   LaserEnd_Ext()
   LIN {X -2.280, Y -28.706, Z 16.150}
   LaserStart_Ext()
   LIN {X -2.280, Y -30.758, Z 16.150}
   LaserEnd_Ext()
   LIN {X -1.280, Y -30.373, Z 16.150}
   LaserStart_Ext()
   LIN {X -1.280, Y -28.244, Z 16.150}
   LaserEnd_Ext()
   LIN {X -1.280, Y -17.881, Z 16.150}
   LaserStart_Ext()
   LIN {X -1.280, Y 7.950, Z 16.150}
   LaserEnd_Ext()
   LIN {X -1.280, Y 30.841, Z 16.150}
   LaserStart_Ext()
   LIN {X -1.280, Y 40.883, Z 16.150}
   LaserEnd_Ext()
   LIN {X -0.280, Y 41.227, Z 16.150}
   LaserStart_Ext()
   LIN {X -0.280, Y -18.756, Z 16.150}
   LaserEnd_Ext()
   LIN {X -0.280, Y -27.386, Z 16.150}
   LaserStart_Ext()
   LIN {X -0.280, Y -29.936, Z 16.150}
   LaserEnd_Ext()
   LIN {X 0.720, Y -29.192, Z 16.150}
   LaserStart_Ext()
   LIN {X 0.720, Y -26.394, Z 16.150}
   LaserEnd_Ext()
   LIN {X 0.720, Y -19.688, Z 16.150}
   LaserStart_Ext()
   LIN {X 0.720, Y 41.215, Z 16.150}
   LaserEnd_Ext()
   LIN {X 1.720, Y 40.867, Z 16.150}
   LaserStart_Ext()
   LIN {X 1.720, Y -23.022, Z 16.150}
   LaserEnd_Ext()
   LIN {X 1.720, Y -23.653, Z 16.150}
   LaserStart_Ext()
   LIN {X 1.720, Y -28.282, Z 16.150}
   LaserEnd_Ext()
   LIN {X 2.720, Y -26.691, Z 16.150}
   LaserStart_Ext()
   LIN {X 2.720, Y 39.894, Z 16.150}
   LaserEnd_Ext()
   LIN {X 3.720, Y 37.137, Z 16.150}
   LaserStart_Ext()
   LIN {X 3.720, Y -24.352, Z 16.150}
   LaserEnd_Ext()
   LIN {X 4.720, Y -20.713, Z 16.150}
   LaserStart_Ext()
   LIN {X 4.720, Y 33.485, Z 16.150}
   LaserEnd_Ext()
   LIN {X 5.720, Y 29.196, Z 16.150}
   LaserStart_Ext()
   LIN {X 5.720, Y -16.461, Z 16.150}
   LaserEnd_Ext()
   LIN {X 6.720, Y -11.133, Z 16.150}
   LaserStart_Ext()
   LIN {X 6.720, Y 23.723, Z 16.150}
   LaserEnd_Ext()
   LIN {X 7.720, Y 15.659, Z 16.150}
   LaserStart_Ext()
   LIN {X 7.720, Y -3.019, Z 16.150}
   LaserEnd_Ext()
   LIN {X -5.450, Y -18.220, Z 17.000}
   LaserStart_Ext()
   LIN {X -4.243, Y -18.029, Z 17.000} C_DIS
   LIN {X -3.691, Y -18.103, Z 17.000} C_DIS
   LIN {X -1.993, Y -18.493, Z 17.000} C_DIS
   LIN {X -0.415, Y -19.723, Z 17.000} C_DIS
   LIN {X -0.294, Y -19.833, Z 17.000} C_DIS
   LIN {X 0.476, Y -21.132, Z 17.000} C_DIS
   LIN {X 0.538, Y -21.297, Z 17.000} C_DIS
   LIN {X 0.796, Y -22.497, Z 17.000} C_DIS
   LIN {X 0.823, Y -23.103, Z 17.000} C_DIS
   LIN {X 0.725, Y -23.910, Z 17.000} C_DIS
   LIN {X 0.164, Y -25.394, Z 17.000} C_DIS
   LIN {X -0.518, Y -26.215, Z 17.000} C_DIS
   LIN {X -2.057, Y -27.540, Z 17.000} C_DIS
   LIN {X -3.374, Y -27.928, Z 17.000} C_DIS
   LIN {X -3.846, Y -28.000, Z 17.000} C_DIS
   LIN {X -4.662, Y -27.994, Z 17.000} C_DIS
   LIN {X -5.636, Y -27.809, Z 17.000} C_DIS
   LIN {X -6.024, Y -27.663, Z 17.000} C_DIS
   LIN {X -6.355, Y -27.534, Z 17.000} C_DIS
   LIN {X -6.753, Y -27.306, Z 17.000} C_DIS
   LIN {X -6.978, Y -27.176, Z 17.000} C_DIS
   LIN {X -7.114, Y -27.065, Z 17.000} C_DIS
   LIN {X -7.700, Y -26.583, Z 17.000} C_DIS
   LIN {X -7.930, Y -26.330, Z 17.000} C_DIS
   LIN {X -8.121, Y -26.097, Z 17.000} C_DIS
   LIN {X -8.706, Y -25.137, Z 17.000} C_DIS
   LIN {X -8.894, Y -24.608, Z 17.000} C_DIS
   LIN {X -9.152, Y -23.495, Z 17.000} C_DIS
   LIN {X -9.139, Y -22.986, Z 17.000} C_DIS
   LIN {X -8.912, Y -21.521, Z 17.000} C_DIS
   LIN {X -8.559, Y -20.716, Z 17.000} C_DIS
   LIN {X -7.683, Y -19.537, Z 17.000} C_DIS
   LIN {X -6.841, Y -18.853, Z 17.000} C_DIS
   LIN {X -5.450, Y -18.220, Z 17.000}
   LaserEnd_Ext()
   LIN {X 6.431, Y 30.497, Z 17.000}
   LaserStart_Ext()
   LIN {X 6.704, Y 29.214, Z 17.000} C_DIS
   LIN {X 6.976, Y 27.929, Z 17.000} C_DIS
   LIN {X 7.359, Y 25.908, Z 17.000} C_DIS
   LIN {X 8.015, Y 21.716, Z 17.000} C_DIS
   LIN {X 8.202, Y 20.509, Z 17.000} C_DIS
   LIN {X 8.387, Y 18.945, Z 17.000} C_DIS
   LIN {X 8.618, Y 16.899, Z 17.000} C_DIS
   LIN {X 8.905, Y 13.181, Z 17.000} C_DIS
   LIN {X 8.966, Y 12.376, Z 17.000} C_DIS
   LIN {X 8.983, Y 11.912, Z 17.000} C_DIS
   LIN {X 9.122, Y 8.334, Z 17.000} C_DIS
   LIN {X 9.128, Y 6.206, Z 17.000} C_DIS
   LIN {X 8.999, Y 1.165, Z 17.000} C_DIS
   LIN {X 8.973, Y 0.207, Z 17.000} C_DIS
   LIN {X 8.911, Y -0.907, Z 17.000} C_DIS
   LIN {X 8.854, Y -1.635, Z 17.000} C_DIS
   LIN {X 8.591, Y -4.753, Z 17.000} C_DIS
   LIN {X 8.449, Y -6.070, Z 17.000} C_DIS
   LIN {X 7.879, Y -10.311, Z 17.000} C_DIS
   LIN {X 7.784, Y -11.041, Z 17.000} C_DIS
   LIN {X 7.748, Y -11.256, Z 17.000} C_DIS
   LIN {X 6.863, Y -16.094, Z 17.000} C_DIS
   LIN {X 6.582, Y -17.401, Z 17.000} C_DIS
   LIN {X 6.121, Y -19.432, Z 17.000} C_DIS
   LIN {X 5.403, Y -22.271, Z 17.000} C_DIS
   LIN {X 5.365, Y -22.424, Z 17.000} C_DIS
   LIN {X 5.334, Y -22.533, Z 17.000} C_DIS
   LIN {X 4.475, Y -25.565, Z 17.000} C_DIS
   LIN {X 3.364, Y -27.741, Z 17.000} C_DIS
   LIN {X 2.947, Y -28.512, Z 17.000} C_DIS
   LIN {X 1.982, Y -29.389, Z 17.000} C_DIS
   LIN {X 0.757, Y -30.538, Z 17.000} C_DIS
   LIN {X -0.229, Y -30.945, Z 17.000} C_DIS
   LIN {X -2.032, Y -31.734, Z 17.000} C_DIS
   LIN {X -3.925, Y -31.970, Z 17.000} C_DIS
   LIN {X -4.873, Y -31.993, Z 17.000} C_DIS
   LIN {X -6.446, Y -31.592, Z 17.000} C_DIS
   LIN {X -7.400, Y -31.424, Z 17.000} C_DIS
   LIN {X -8.236, Y -31.065, Z 17.000} C_DIS
   LIN {X -10.230, Y -29.705, Z 17.000} C_DIS
   LIN {X -10.335, Y -29.619, Z 17.000} C_DIS
   LIN {X -11.087, Y -28.763, Z 17.000} C_DIS
   LIN {X -11.881, Y -27.714, Z 17.000} C_DIS
   LIN {X -12.470, Y -26.319, Z 17.000} C_DIS
   LIN {X -12.951, Y -25.071, Z 17.000} C_DIS
   LIN {X -12.992, Y -22.192, Z 17.000} C_DIS
   LIN {X -13.010, Y -21.360, Z 17.000} C_DIS
   LIN {X -12.637, Y -20.382, Z 17.000} C_DIS
   LIN {X -11.872, Y -18.401, Z 17.000} C_DIS
   LIN {X -10.989, Y -16.874, Z 17.000} C_DIS
   LIN {X -10.294, Y -15.649, Z 17.000} C_DIS
   LIN {X -9.408, Y -13.978, Z 17.000} C_DIS
   LIN {X -8.733, Y -12.580, Z 17.000} C_DIS
   LIN {X -7.443, Y -9.834, Z 17.000} C_DIS
   LIN {X -6.328, Y -7.025, Z 17.000} C_DIS
   LIN {X -5.522, Y -4.924, Z 17.000} C_DIS
   LIN {X -3.659, Y 1.357, Z 17.000} C_DIS
   LIN {X -3.421, Y 2.167, Z 17.000} C_DIS
   LIN {X -3.273, Y 2.842, Z 17.000} C_DIS
   LIN {X -2.380, Y 7.329, Z 17.000} C_DIS
   LIN {X -2.004, Y 9.910, Z 17.000} C_DIS
   LIN {X -1.776, Y 11.764, Z 17.000} C_DIS
   LIN {X -1.634, Y 13.471, Z 17.000} C_DIS
   LIN {X -1.612, Y 14.054, Z 17.000} C_DIS
   LIN {X -1.468, Y 16.030, Z 17.000} C_DIS
   LIN {X -1.421, Y 19.052, Z 17.000} C_DIS
   LIN {X -1.420, Y 21.163, Z 17.000} C_DIS
   LIN {X -1.595, Y 24.213, Z 17.000} C_DIS
   LIN {X -1.701, Y 25.882, Z 17.000} C_DIS
   LIN {X -2.078, Y 29.186, Z 17.000} C_DIS
   LIN {X -2.124, Y 29.535, Z 17.000} C_DIS
   LIN {X -2.430, Y 31.414, Z 17.000} C_DIS
   LIN {X -2.576, Y 32.326, Z 17.000} C_DIS
   LIN {X -2.668, Y 32.796, Z 17.000} C_DIS
   LIN {X -3.038, Y 34.652, Z 17.000} C_DIS
   LIN {X -3.348, Y 36.019, Z 17.000} C_DIS
   LIN {X -3.393, Y 36.213, Z 17.000} C_DIS
   LIN {X -3.459, Y 36.487, Z 17.000} C_DIS
   LIN {X -3.686, Y 37.429, Z 17.000} C_DIS
   LIN {X -3.738, Y 38.177, Z 17.000} C_DIS
   LIN {X -3.792, Y 38.908, Z 17.000} C_DIS
   LIN {X -3.532, Y 39.736, Z 17.000} C_DIS
   LIN {X -3.360, Y 40.291, Z 17.000} C_DIS
   LIN {X -3.041, Y 40.696, Z 17.000} C_DIS
   LIN {X -2.467, Y 41.418, Z 17.000} C_DIS
   LIN {X -1.848, Y 41.803, Z 17.000} C_DIS
   LIN {X 0.138, Y 42.387, Z 17.000} C_DIS
   LIN {X 0.378, Y 42.367, Z 17.000} C_DIS
   LIN {X 1.926, Y 41.986, Z 17.000} C_DIS
   LIN {X 2.718, Y 41.349, Z 17.000} C_DIS
   LIN {X 3.282, Y 40.891, Z 17.000} C_DIS
   LIN {X 3.746, Y 40.020, Z 17.000} C_DIS
   LIN {X 3.975, Y 39.590, Z 17.000} C_DIS
   LIN {X 4.075, Y 39.268, Z 17.000} C_DIS
   LIN {X 4.413, Y 38.171, Z 17.000} C_DIS
   LIN {X 4.920, Y 36.437, Z 17.000} C_DIS
   LIN {X 4.951, Y 36.329, Z 17.000} C_DIS
   LIN {X 5.025, Y 36.053, Z 17.000} C_DIS
   LIN {X 5.675, Y 33.640, Z 17.000} C_DIS
   LIN {X 6.024, Y 32.202, Z 17.000} C_DIS
   LIN {X 6.431, Y 30.497, Z 17.000}
   LaserEnd_Ext()
   LIN {X -1.387, Y -30.360, Z 17.000}
   LaserStart_Ext()
   LIN {X -7.343, Y -30.360, Z 17.000}
   LaserEnd_Ext()
   LIN {X -8.961, Y -29.360, Z 17.000}
   LaserStart_Ext()
   LIN {X 0.552, Y -29.360, Z 17.000}
   LaserEnd_Ext()
   LIN {X 1.628, Y -28.360, Z 17.000}
   LaserStart_Ext()
   LIN {X -1.486, Y -28.360, Z 17.000}
   LaserEnd_Ext()
   LIN {X -6.925, Y -28.360, Z 17.000}
   LaserStart_Ext()
   LIN {X -10.110, Y -28.360, Z 17.000}
   LaserEnd_Ext()
   LIN {X -10.895, Y -27.360, Z 17.000}
   LaserStart_Ext()
   LIN {X -8.329, Y -27.360, Z 17.000}
   LaserEnd_Ext()
   LIN {X -0.316, Y -27.360, Z 17.000}
   LaserStart_Ext()
   LIN {X 2.433, Y -27.360, Z 17.000}
   LaserEnd_Ext()
   LIN {X 2.946, Y -26.360, Z 17.000}
   LaserStart_Ext()
   LIN {X 0.661, Y -26.360, Z 17.000}
   LaserEnd_Ext()
   LIN {X -9.132, Y -26.360, Z 17.000}
   LaserStart_Ext()
   LIN {X -11.367, Y -26.360, Z 17.000}
   LaserEnd_Ext()
   LIN {X -11.767, Y -25.360, Z 17.000}
   LaserStart_Ext()
   LIN {X -9.688, Y -25.360, Z 17.000}
   LaserEnd_Ext()
   LIN {X 1.246, Y -25.360, Z 17.000}
   LaserStart_Ext()
   LIN {X 3.457, Y -25.360, Z 17.000}
   LaserEnd_Ext()
   LIN {X 3.777, Y -24.360, Z 17.000}
   LaserStart_Ext()
   LIN {X 1.624, Y -24.360, Z 17.000}
   LaserEnd_Ext()
   LIN {X -9.978, Y -24.360, Z 17.000}
   LaserStart_Ext()
   LIN {X -11.961, Y -24.360, Z 17.000}
   LaserEnd_Ext()
   LIN {X -11.975, Y -23.360, Z 17.000}
   LaserStart_Ext()
   LIN {X -10.149, Y -23.360, Z 17.000}
   LaserEnd_Ext()
   LIN {X 1.799, Y -23.360, Z 17.000}
   LaserStart_Ext()
   LIN {X 4.061, Y -23.360, Z 17.000}
   LaserEnd_Ext()
   LIN {X 4.344, Y -22.360, Z 17.000}
   LaserStart_Ext()
   LIN {X 1.786, Y -22.360, Z 17.000}
   LaserEnd_Ext()
   LIN {X -10.054, Y -22.360, Z 17.000}
   LaserStart_Ext()
   LIN {X -11.990, Y -22.360, Z 17.000}
   LaserEnd_Ext()
   LIN {X -11.940, Y -21.360, Z 17.000}
   LaserStart_Ext()
   LIN {X -9.899, Y -21.360, Z 17.000}
   LaserEnd_Ext()
   LIN {X 1.575, Y -21.360, Z 17.000}
   LaserStart_Ext()
   LIN {X 4.602, Y -21.360, Z 17.000}
   LaserEnd_Ext()
   LIN {X 4.855, Y -20.360, Z 17.000}
   LaserStart_Ext()
   LIN {X 1.181, Y -20.360, Z 17.000}
   LaserEnd_Ext()
   LIN {X -9.495, Y -20.360, Z 17.000}
   LaserStart_Ext()
   LIN {X -11.557, Y -20.360, Z 17.000}
   LaserEnd_Ext()
   LIN {X -11.171, Y -19.360, Z 17.000}
   LaserStart_Ext()
   LIN {X -8.797, Y -19.360, Z 17.000}
   LaserEnd_Ext()
   LIN {X 0.589, Y -19.360, Z 17.000}
   LaserStart_Ext()
   LIN {X 5.108, Y -19.360, Z 17.000}
   LaserEnd_Ext()
   LIN {X 5.339, Y -18.360, Z 17.000}
   LaserStart_Ext()
   LIN {X -0.537, Y -18.360, Z 17.000}
   LaserEnd_Ext()
   LIN {X -7.820, Y -18.360, Z 17.000}
   LaserStart_Ext()
   LIN {X -10.693, Y -18.360, Z 17.000}
   LaserEnd_Ext()
   LIN {X -10.115, Y -17.360, Z 17.000}
   LaserStart_Ext()
   LIN {X -5.975, Y -17.360, Z 17.000}
   LaserEnd_Ext()
   LIN {X -2.459, Y -17.360, Z 17.000}
   LaserStart_Ext()
   LIN {X 5.566, Y -17.360, Z 17.000}
   LaserEnd_Ext()
   LIN {X 5.783, Y -16.360, Z 17.000}
   LaserStart_Ext()
   LIN {X -9.548, Y -16.360, Z 17.000}
   LaserEnd_Ext()
   LIN {X -9.009, Y -15.360, Z 17.000}
   LaserStart_Ext()
   LIN {X 5.981, Y -15.360, Z 17.000}
   LaserEnd_Ext()
   LIN {X 6.163, Y -14.360, Z 17.000}
   LaserStart_Ext()
   LIN {X -8.482, Y -14.360, Z 17.000}
   LaserEnd_Ext()
   LIN {X -7.999, Y -13.360, Z 17.000}
   LaserStart_Ext()
   LIN {X 6.346, Y -13.360, Z 17.000}
   LaserEnd_Ext()
   LIN {X 6.529, Y -12.360, Z 17.000}
   LaserStart_Ext()
   LIN {X -7.525, Y -12.360, Z 17.000}
   LaserEnd_Ext()
   LIN {X -7.055, Y -11.360, Z 17.000}
   LaserStart_Ext()
   LIN {X 6.712, Y -11.360, Z 17.000}
   LaserEnd_Ext()
   LIN {X 6.864, Y -10.360, Z 17.000}
   LaserStart_Ext()
   LIN {X -6.585, Y -10.360, Z 17.000}
   LaserEnd_Ext()
   LIN {X -6.179, Y -9.360, Z 17.000}
   LaserStart_Ext()
   LIN {X 6.998, Y -9.360, Z 17.000}
   LaserEnd_Ext()
   LIN {X 7.132, Y -8.360, Z 17.000}
   LaserStart_Ext()
   LIN {X -5.782, Y -8.360, Z 17.000}
   LaserEnd_Ext()
   LIN {X -5.385, Y -7.360, Z 17.000}
   LaserStart_Ext()
   LIN {X 7.267, Y -7.360, Z 17.000}
   LaserEnd_Ext()
   LIN {X 7.401, Y -6.360, Z 17.000}
   LaserStart_Ext()
   LIN {X -5.002, Y -6.360, Z 17.000}
   LaserEnd_Ext()
   LIN {X -4.619, Y -5.360, Z 17.000}
   LaserStart_Ext()
   LIN {X 7.520, Y -5.360, Z 17.000}
   LaserEnd_Ext()
   LIN {X 7.621, Y -4.360, Z 17.000}
   LaserStart_Ext()
   LIN {X -4.312, Y -4.360, Z 17.000}
   LaserEnd_Ext()
   LIN {X -4.015, Y -3.360, Z 17.000}
   LaserStart_Ext()
   LIN {X 7.705, Y -3.360, Z 17.000}
   LaserEnd_Ext()
   LIN {X 7.790, Y -2.360, Z 17.000}
   LaserStart_Ext()
   LIN {X -3.718, Y -2.360, Z 17.000}
   LaserEnd_Ext()
   LIN {X -3.422, Y -1.360, Z 17.000}
   LaserStart_Ext()
   LIN {X 7.873, Y -1.360, Z 17.000}
   LaserEnd_Ext()
   LIN {X 7.940, Y -0.360, Z 17.000}
   LaserStart_Ext()
   LIN {X -3.125, Y -0.360, Z 17.000}
   LaserEnd_Ext()
   LIN {X -2.828, Y 0.640, Z 17.000}
   LaserStart_Ext()
   LIN {X 7.984, Y 0.640, Z 17.000}
   LaserEnd_Ext()
   LIN {X 8.011, Y 1.640, Z 17.000}
   LaserStart_Ext()
   LIN {X -2.534, Y 1.640, Z 17.000}
   LaserEnd_Ext()
   LIN {X -2.294, Y 2.640, Z 17.000}
   LaserStart_Ext()
   LIN {X 8.037, Y 2.640, Z 17.000}
   LaserEnd_Ext()
   LIN {X 8.062, Y 3.640, Z 17.000}
   LaserStart_Ext()
   LIN {X -2.095, Y 3.640, Z 17.000}
   LaserEnd_Ext()
   LIN {X -1.896, Y 4.640, Z 17.000}
   LaserStart_Ext()
   LIN {X 8.087, Y 4.640, Z 17.000}
   LaserEnd_Ext()
   LIN {X 8.113, Y 5.640, Z 17.000}
   LaserStart_Ext()
   LIN {X -1.697, Y 5.640, Z 17.000}
   LaserEnd_Ext()
   LIN {X -1.497, Y 6.640, Z 17.000}
   LaserStart_Ext()
   LIN {X 8.126, Y 6.640, Z 17.000}
   LaserEnd_Ext()
   LIN {X 8.124, Y 7.640, Z 17.000}
   LaserStart_Ext()
   LIN {X -1.324, Y 7.640, Z 17.000}
   LaserEnd_Ext()
   LIN {X -1.178, Y 8.640, Z 17.000}
   LaserStart_Ext()
   LIN {X 8.109, Y 8.640, Z 17.000}
   LaserEnd_Ext()
   LIN {X 8.070, Y 9.640, Z 17.000}
   LaserStart_Ext()
   LIN {X -1.033, Y 9.640, Z 17.000}
   LaserEnd_Ext()
   LIN {X -0.907, Y 10.640, Z 17.000}
   LaserStart_Ext()
   LIN {X 8.031, Y 10.640, Z 17.000}
   LaserEnd_Ext()
   LIN {X 7.993, Y 11.640, Z 17.000}
   LaserStart_Ext()
   LIN {X -0.783, Y 11.640, Z 17.000}
   LaserEnd_Ext()
   LIN {X -0.700, Y 12.640, Z 17.000}
   LaserStart_Ext()
   LIN {X 7.943, Y 12.640, Z 17.000}
   LaserEnd_Ext()
   LIN {X 7.867, Y 13.640, Z 17.000}
   LaserStart_Ext()
   LIN {X -0.627, Y 13.640, Z 17.000}
   LaserEnd_Ext()
   LIN {X -0.567, Y 14.640, Z 17.000}
   LaserStart_Ext()
   LIN {X 7.790, Y 14.640, Z 17.000}
   LaserEnd_Ext()
   LIN {X 7.713, Y 15.640, Z 17.000}
   LaserStart_Ext()
   LIN {X -0.494, Y 15.640, Z 17.000}
   LaserEnd_Ext()
   LIN {X -0.459, Y 16.640, Z 17.000}
   LaserStart_Ext()
   LIN {X 7.635, Y 16.640, Z 17.000}
   LaserEnd_Ext()
   LIN {X 7.528, Y 17.640, Z 17.000}
   LaserStart_Ext()
   LIN {X -0.443, Y 17.640, Z 17.000}
   LaserEnd_Ext()
   LIN {X -0.427, Y 18.640, Z 17.000}
   LaserStart_Ext()
   LIN {X 7.415, Y 18.640, Z 17.000}
   LaserEnd_Ext()
   LIN {X 7.298, Y 19.640, Z 17.000}
   LaserStart_Ext()
   LIN {X -0.420, Y 19.640, Z 17.000}
   LaserEnd_Ext()
   LIN {X -0.420, Y 20.640, Z 17.000}
   LaserStart_Ext()
   LIN {X 7.169, Y 20.640, Z 17.000}
   LaserEnd_Ext()
   LIN {X 7.015, Y 21.640, Z 17.000}
   LaserStart_Ext()
   LIN {X -0.446, Y 21.640, Z 17.000}
   LaserEnd_Ext()
   LIN {X -0.503, Y 22.640, Z 17.000}
   LaserStart_Ext()
   LIN {X 6.858, Y 22.640, Z 17.000}
   LaserEnd_Ext()
   LIN {X 6.702, Y 23.640, Z 17.000}
   LaserStart_Ext()
   LIN {X -0.560, Y 23.640, Z 17.000}
   LaserEnd_Ext()
   LIN {X -0.620, Y 24.640, Z 17.000}
   LaserStart_Ext()
   LIN {X 6.545, Y 24.640, Z 17.000}
   LaserEnd_Ext()
   LIN {X 6.389, Y 25.640, Z 17.000}
   LaserStart_Ext()
   LIN {X -0.684, Y 25.640, Z 17.000}
   LaserEnd_Ext()
   LIN {X -0.781, Y 26.640, Z 17.000}
   LaserStart_Ext()
   LIN {X 6.202, Y 26.640, Z 17.000}
   LaserEnd_Ext()
   LIN {X 6.013, Y 27.640, Z 17.000}
   LaserStart_Ext()
   LIN {X -0.895, Y 27.640, Z 17.000}
   LaserEnd_Ext()
   LIN {X -1.009, Y 28.640, Z 17.000}
   LaserStart_Ext()
   LIN {X 5.803, Y 28.640, Z 17.000}
   LaserEnd_Ext()
   LIN {X 5.591, Y 29.640, Z 17.000}
   LaserStart_Ext()
   LIN {X -1.130, Y 29.640, Z 17.000}
   LaserEnd_Ext()
   LIN {X -1.291, Y 30.640, Z 17.000}
   LaserStart_Ext()
   LIN {X 5.368, Y 30.640, Z 17.000}
   LaserEnd_Ext()
   LIN {X 5.130, Y 31.640, Z 17.000}
   LaserStart_Ext()
   LIN {X -1.453, Y 31.640, Z 17.000}
   LaserEnd_Ext()
   LIN {X -1.619, Y 32.640, Z 17.000}
   LaserStart_Ext()
   LIN {X 4.888, Y 32.640, Z 17.000}
   LaserEnd_Ext()
   LIN {X 4.639, Y 33.640, Z 17.000}
   LaserStart_Ext()
   LIN {X -1.817, Y 33.640, Z 17.000}
   LaserEnd_Ext()
   LIN {X -2.016, Y 34.640, Z 17.000}
   LaserStart_Ext()
   LIN {X 4.370, Y 34.640, Z 17.000}
   LaserEnd_Ext()
   LIN {X 4.101, Y 35.640, Z 17.000}
   LaserStart_Ext()
   LIN {X -2.237, Y 35.640, Z 17.000}
   LaserEnd_Ext()
   LIN {X -2.467, Y 36.640, Z 17.000}
   LaserStart_Ext()
   LIN {X 3.819, Y 36.640, Z 17.000}
   LaserEnd_Ext()
   LIN {X 3.527, Y 37.640, Z 17.000}
   LaserStart_Ext()
   LIN {X -2.699, Y 37.640, Z 17.000}
   LaserEnd_Ext()
   LIN {X -2.769, Y 38.640, Z 17.000}
   LaserStart_Ext()
   LIN {X 3.223, Y 38.640, Z 17.000}
   LaserEnd_Ext()
   LIN {X 2.815, Y 39.640, Z 17.000}
   LaserStart_Ext()
   LIN {X -2.515, Y 39.640, Z 17.000}
   LaserEnd_Ext()
   LIN {X -1.808, Y 40.640, Z 17.000}
   LaserStart_Ext()
   LIN {X 2.004, Y 40.640, Z 17.000}
   LaserEnd_Ext()
   LIN {X -7.199, Y -26.888, Z 17.850}
   LaserStart_Ext()
   LIN {X -7.951, Y -26.121, Z 17.850} C_DIS
   LIN {X -8.282, Y -25.717, Z 17.850} C_DIS
   LIN {X -8.483, Y -25.388, Z 17.850} C_DIS
   LIN {X -8.955, Y -24.057, Z 17.850} C_DIS
   LIN {X -9.064, Y -23.586, Z 17.850} C_DIS
   LIN {X -9.035, Y -22.414, Z 17.850} C_DIS
   LIN {X -8.949, Y -21.857, Z 17.850} C_DIS
   LIN {X -8.225, Y -20.211, Z 17.850} C_DIS
   LIN {X -7.965, Y -19.859, Z 17.850} C_DIS
   LIN {X -6.391, Y -18.581, Z 17.850} C_DIS
   LIN {X -5.723, Y -18.277, Z 17.850} C_DIS
   LIN {X -4.882, Y -18.144, Z 17.850} C_DIS
   LIN {X -4.003, Y -17.970, Z 17.850} C_DIS
   LIN {X -2.911, Y -18.217, Z 17.850} C_DIS
   LIN {X -1.929, Y -18.443, Z 17.850} C_DIS
   LIN {X -1.244, Y -18.977, Z 17.850} C_DIS
   LIN {X -0.251, Y -19.745, Z 17.850} C_DIS
   LIN {X 0.332, Y -20.733, Z 17.850} C_DIS
   LIN {X 0.634, Y -21.329, Z 17.850} C_DIS
   LIN {X 0.905, Y -22.765, Z 17.850} C_DIS
   LIN {X 0.889, Y -22.915, Z 17.850} C_DIS
   LIN {X 0.735, Y -24.187, Z 17.850} C_DIS
   LIN {X 0.502, Y -24.803, Z 17.850} C_DIS
   LIN {X -1.041, Y -26.660, Z 17.850} C_DIS
   LIN {X -2.040, Y -27.520, Z 17.850} C_DIS
   LIN {X -3.518, Y -27.921, Z 17.850} C_DIS
   LIN {X -3.698, Y -27.945, Z 17.850} C_DIS
   LIN {X -5.347, Y -27.820, Z 17.850} C_DIS
   LIN {X -5.523, Y -27.764, Z 17.850} C_DIS
   LIN {X -6.270, Y -27.494, Z 17.850} C_DIS
   LIN {X -6.726, Y -27.234, Z 17.850} C_DIS
   LIN {X -6.894, Y -27.138, Z 17.850} C_DIS
   LIN {X -7.199, Y -26.888, Z 17.850}
   LaserEnd_Ext()
   LIN {X -12.607, Y -25.739, Z 17.850}
   LaserStart_Ext()
   LIN {X -12.874, Y -25.045, Z 17.850} C_DIS
   LIN {X -12.897, Y -23.443, Z 17.850} C_DIS
   LIN {X -12.942, Y -21.334, Z 17.850} C_DIS
   LIN {X -11.997, Y -18.854, Z 17.850} C_DIS
   LIN {X -11.811, Y -18.372, Z 17.850} C_DIS
   LIN {X -11.596, Y -18.001, Z 17.850} C_DIS
   LIN {X -10.144, Y -15.439, Z 17.850} C_DIS
   LIN {X -9.520, Y -14.262, Z 17.850} C_DIS
   LIN {X -8.527, Y -12.209, Z 17.850} C_DIS
   LIN {X -7.477, Y -9.972, Z 17.850} C_DIS
   LIN {X -6.032, Y -6.333, Z 17.850} C_DIS
   LIN {X -5.652, Y -5.341, Z 17.850} C_DIS
   LIN {X -4.084, Y -0.057, Z 17.850} C_DIS
   LIN {X -3.441, Y 2.074, Z 17.850} C_DIS
   LIN {X -3.383, Y 2.320, Z 17.850} C_DIS
   LIN {X -3.232, Y 3.117, Z 17.850} C_DIS
   LIN {X -2.341, Y 7.589, Z 17.850} C_DIS
   LIN {X -2.089, Y 9.319, Z 17.850} C_DIS
   LIN {X -1.785, Y 11.782, Z 17.850} C_DIS
   LIN {X -1.695, Y 12.878, Z 17.850} C_DIS
   LIN {X -1.681, Y 13.252, Z 17.850} C_DIS
   LIN {X -1.501, Y 15.721, Z 17.850} C_DIS
   LIN {X -1.441, Y 19.497, Z 17.850} C_DIS
   LIN {X -1.441, Y 20.949, Z 17.850} C_DIS
   LIN {X -1.561, Y 23.046, Z 17.850} C_DIS
   LIN {X -1.753, Y 26.053, Z 17.850} C_DIS
   LIN {X -2.052, Y 28.678, Z 17.850} C_DIS
   LIN {X -2.191, Y 29.720, Z 17.850} C_DIS
   LIN {X -2.349, Y 30.693, Z 17.850} C_DIS
   LIN {X -2.630, Y 32.375, Z 17.850} C_DIS
   LIN {X -3.021, Y 34.319, Z 17.850} C_DIS
   LIN {X -3.097, Y 34.700, Z 17.850} C_DIS
   LIN {X -3.138, Y 34.878, Z 17.850} C_DIS
   LIN {X -3.456, Y 36.260, Z 17.850} C_DIS
   LIN {X -3.655, Y 37.082, Z 17.850} C_DIS
   LIN {X -3.752, Y 37.476, Z 17.850} C_DIS
   LIN {X -3.805, Y 38.195, Z 17.850} C_DIS
   LIN {X -3.860, Y 38.954, Z 17.850} C_DIS
   LIN {X -3.673, Y 39.552, Z 17.850} C_DIS
   LIN {X -3.417, Y 40.366, Z 17.850} C_DIS
   LIN {X -2.874, Y 41.048, Z 17.850} C_DIS
   LIN {X -2.540, Y 41.468, Z 17.850} C_DIS
   LIN {X -2.371, Y 41.573, Z 17.850} C_DIS
   LIN {X -1.764, Y 41.752, Z 17.850} C_DIS
   LIN {X 0.151, Y 42.459, Z 17.850} C_DIS
   LIN {X 1.373, Y 42.163, Z 17.850} C_DIS
   LIN {X 1.849, Y 42.046, Z 17.850} C_DIS
   LIN {X 2.427, Y 41.580, Z 17.850} C_DIS
   LIN {X 3.208, Y 40.954, Z 17.850} C_DIS
   LIN {X 3.517, Y 40.381, Z 17.850} C_DIS
   LIN {X 3.904, Y 39.655, Z 17.850} C_DIS
   LIN {X 4.262, Y 38.506, Z 17.850} C_DIS
   LIN {X 4.346, Y 38.237, Z 17.850} C_DIS
   LIN {X 4.412, Y 38.014, Z 17.850} C_DIS
   LIN {X 4.888, Y 36.396, Z 17.850} C_DIS
   LIN {X 5.409, Y 34.486, Z 17.850} C_DIS
   LIN {X 5.618, Y 33.709, Z 17.850} C_DIS
   LIN {X 6.063, Y 31.872, Z 17.850} C_DIS
   LIN {X 6.388, Y 30.538, Z 17.850} C_DIS
   LIN {X 6.530, Y 29.855, Z 17.850} C_DIS
   LIN {X 7.077, Y 27.267, Z 17.850} C_DIS
   LIN {X 7.293, Y 26.129, Z 17.850} C_DIS
   LIN {X 8.229, Y 20.144, Z 17.850} C_DIS
   LIN {X 8.261, Y 19.939, Z 17.850} C_DIS
   LIN {X 8.293, Y 19.672, Z 17.850} C_DIS
   LIN {X 8.616, Y 16.808, Z 17.850} C_DIS
   LIN {X 8.902, Y 13.104, Z 17.850} C_DIS
   LIN {X 8.962, Y 12.366, Z 17.850} C_DIS
   LIN {X 8.993, Y 11.606, Z 17.850} C_DIS
   LIN {X 9.129, Y 8.117, Z 17.850} C_DIS
   LIN {X 9.133, Y 6.586, Z 17.850} C_DIS
   LIN {X 8.963, Y -0.111, Z 17.850} C_DIS
   LIN {X 8.953, Y -0.469, Z 17.850} C_DIS
   LIN {X 8.930, Y -0.886, Z 17.850} C_DIS
   LIN {X 8.908, Y -1.158, Z 17.850} C_DIS
   LIN {X 8.543, Y -5.485, Z 17.850} C_DIS
   LIN {X 8.531, Y -5.595, Z 17.850} C_DIS
   LIN {X 8.484, Y -5.949, Z 17.850} C_DIS
   LIN {X 7.844, Y -10.867, Z 17.850} C_DIS
   LIN {X 7.600, Y -12.315, Z 17.850} C_DIS
   LIN {X 6.948, Y -15.881, Z 17.850} C_DIS
   LIN {X 6.424, Y -18.316, Z 17.850} C_DIS
   LIN {X 6.211, Y -19.254, Z 17.850} C_DIS
   LIN {X 5.879, Y -20.567, Z 17.850} C_DIS
   LIN {X 5.436, Y -22.356, Z 17.850} C_DIS
   LIN {X 5.083, Y -23.629, Z 17.850} C_DIS
   LIN {X 4.553, Y -25.498, Z 17.850} C_DIS
   LIN {X 3.327, Y -27.899, Z 17.850} C_DIS
   LIN {X 3.092, Y -28.374, Z 17.850} C_DIS
   LIN {X 2.839, Y -28.625, Z 17.850} C_DIS
   LIN {X 0.897, Y -30.446, Z 17.850} C_DIS
   LIN {X -1.260, Y -31.336, Z 17.850} C_DIS
   LIN {X -2.220, Y -31.756, Z 17.850} C_DIS
   LIN {X -3.227, Y -31.882, Z 17.850} C_DIS
   LIN {X -5.000, Y -31.926, Z 17.850} C_DIS
   LIN {X -7.724, Y -31.231, Z 17.850} C_DIS
   LIN {X -7.883, Y -31.154, Z 17.850} C_DIS
   LIN {X -10.100, Y -29.718, Z 17.850} C_DIS
   LIN {X -11.311, Y -28.304, Z 17.850} C_DIS
   LIN {X -11.541, Y -28.042, Z 17.850} C_DIS
   LIN {X -11.753, Y -27.762, Z 17.850} C_DIS
   LIN {X -12.607, Y -25.739, Z 17.850}
   LaserEnd_Ext()
   LIN {X 7.602, Y -4.746, Z 17.850}
   LaserStart_Ext()
   LIN {X 7.602, Y 16.879, Z 17.850}
   LaserEnd_Ext()
   LIN {X 6.602, Y 24.078, Z 17.850}
   LaserStart_Ext()
   LIN {X 6.602, Y -12.212, Z 17.850}
   LaserEnd_Ext()
   LIN {X 5.602, Y -17.382, Z 17.850}
   LaserStart_Ext()
   LIN {X 5.602, Y 29.412, Z 17.850}
   LaserEnd_Ext()
   LIN {X 4.602, Y 33.636, Z 17.850}
   LaserStart_Ext()
   LIN {X 4.602, Y -21.562, Z 17.850}
   LaserEnd_Ext()
   LIN {X 3.602, Y -25.162, Z 17.850}
   LaserStart_Ext()
   LIN {X 3.602, Y 37.225, Z 17.850}
   LaserEnd_Ext()
   LIN {X 2.602, Y 39.970, Z 17.850}
   LaserStart_Ext()
   LIN {X 2.602, Y -27.121, Z 17.850}
   LaserEnd_Ext()
   LIN {X 1.602, Y -28.414, Z 17.850}
   LaserStart_Ext()
   LIN {X 1.602, Y -24.721, Z 17.850}
   LaserEnd_Ext()
   LIN {X 1.602, Y -21.082, Z 17.850}
   LaserStart_Ext()
   LIN {X 1.602, Y 40.961, Z 17.850}
   LaserEnd_Ext()
   LIN {X 0.602, Y 41.321, Z 17.850}
   LaserStart_Ext()
   LIN {X 0.602, Y -19.223, Z 17.850}
   LaserEnd_Ext()
   LIN {X 0.602, Y -26.247, Z 17.850}
   LaserStart_Ext()
   LIN {X 0.602, Y -29.352, Z 17.850}
   LaserEnd_Ext()
   LIN {X -0.398, Y -29.899, Z 17.850}
   LaserStart_Ext()
   LIN {X -0.398, Y -27.426, Z 17.850}
   LaserEnd_Ext()
   LIN {X -0.398, Y -18.367, Z 17.850}
   LaserStart_Ext()
   LIN {X -0.398, Y 41.190, Z 17.850}
   LaserEnd_Ext()
   LIN {X -1.398, Y 40.821, Z 17.850}
   LaserStart_Ext()
   LIN {X -1.398, Y 31.068, Z 17.850}
   LaserEnd_Ext()
   LIN {X -1.398, Y 7.203, Z 17.850}
   LaserStart_Ext()
   LIN {X -1.398, Y -17.596, Z 17.850}
   LaserEnd_Ext()
   LIN {X -1.398, Y -28.286, Z 17.850}
   LaserStart_Ext()
   LIN {X -1.398, Y -30.312, Z 17.850}
   LaserEnd_Ext()
   LIN {X -2.398, Y -30.743, Z 17.850}
   LaserStart_Ext()
   LIN {X -2.398, Y -28.654, Z 17.850}
   LaserEnd_Ext()
   LIN {X -2.398, Y -17.309, Z 17.850}
   LaserStart_Ext()
   LIN {X -2.398, Y 2.144, Z 17.850}
   LaserEnd_Ext()
   LIN {X -2.398, Y 36.124, Z 17.850}
   LaserStart_Ext()
   LIN {X -2.398, Y 40.041, Z 17.850}
   LaserEnd_Ext()
   LIN {X -3.398, Y -1.260, Z 17.850}
   LaserStart_Ext()
   LIN {X -3.398, Y -17.082, Z 17.850}
   LaserEnd_Ext()
   LIN {X -3.398, Y -28.914, Z 17.850}
   LaserStart_Ext()
   LIN {X -3.398, Y -30.886, Z 17.850}
   LaserEnd_Ext()
   LIN {X -4.398, Y -30.911, Z 17.850}
   LaserStart_Ext()
   LIN {X -4.398, Y -28.895, Z 17.850}
   LaserEnd_Ext()
   LIN {X -4.398, Y -17.029, Z 17.850}
   LaserStart_Ext()
   LIN {X -4.398, Y -4.630, Z 17.850}
   LaserEnd_Ext()
   LIN {X -5.398, Y -7.445, Z 17.850}
   LaserStart_Ext()
   LIN {X -5.398, Y -17.213, Z 17.850}
   LaserEnd_Ext()
   LIN {X -5.398, Y -28.819, Z 17.850}
   LaserStart_Ext()
   LIN {X -5.398, Y -30.793, Z 17.850}
   LaserEnd_Ext()
   LIN {X -6.398, Y -30.537, Z 17.850}
   LaserStart_Ext()
   LIN {X -6.398, Y -28.511, Z 17.850}
   LaserEnd_Ext()
   LIN {X -6.398, Y -17.486, Z 17.850}
   LaserStart_Ext()
   LIN {X -6.398, Y -9.965, Z 17.850}
   LaserEnd_Ext()
   LIN {X -7.398, Y -12.157, Z 17.850}
   LaserStart_Ext()
   LIN {X -7.398, Y -18.111, Z 17.850}
   LaserEnd_Ext()
   LIN {X -7.398, Y -28.001, Z 17.850}
   LaserStart_Ext()
   LIN {X -7.398, Y -30.277, Z 17.850}
   LaserEnd_Ext()
   LIN {X -8.398, Y -29.629, Z 17.850}
   LaserStart_Ext()
   LIN {X -8.398, Y -27.094, Z 17.850}
   LaserEnd_Ext()
   LIN {X -8.398, Y -18.923, Z 17.850}
   LaserStart_Ext()
   LIN {X -8.398, Y -14.239, Z 17.850}
   LaserEnd_Ext()
   LIN {X -9.398, Y -16.151, Z 17.850}
   LaserStart_Ext()
   LIN {X -9.398, Y -20.394, Z 17.850}
   LaserEnd_Ext()
   LIN {X -9.398, Y -25.789, Z 17.850}
   LaserStart_Ext()
   LIN {X -9.398, Y -28.981, Z 17.850}
   LaserEnd_Ext()
   LIN {X -10.398, Y -27.833, Z 17.850}
   LaserStart_Ext()
   LIN {X -10.398, Y -17.916, Z 17.850}
   LaserEnd_Ext()
   LIN {X -11.398, Y -20.091, Z 17.850}
   LaserStart_Ext()
   LIN {X -11.398, Y -26.031, Z 17.850}
   LaserEnd_Ext()
   LIN {X -6.544, Y -27.180, Z 18.700}
   LaserStart_Ext()
   LIN {X -8.181, Y -25.705, Z 18.700} C_DIS
   LIN {X -8.410, Y -25.323, Z 18.700} C_DIS
   LIN {X -8.961, Y -23.727, Z 18.700} C_DIS
   LIN {X -8.985, Y -23.561, Z 18.700} C_DIS
   LIN {X -8.954, Y -22.174, Z 18.700} C_DIS
   LIN {X -8.871, Y -21.834, Z 18.700} C_DIS
   LIN {X -8.140, Y -20.130, Z 18.700} C_DIS
   LIN {X -7.946, Y -19.855, Z 18.700} C_DIS
   LIN {X -6.048, Y -18.382, Z 18.700} C_DIS
   LIN {X -5.844, Y -18.301, Z 18.700} C_DIS
   LIN {X -3.940, Y -17.924, Z 18.700} C_DIS
   LIN {X -2.371, Y -18.280, Z 18.700} C_DIS
   LIN {X -1.866, Y -18.392, Z 18.700} C_DIS
   LIN {X -1.387, Y -18.760, Z 18.700} C_DIS
   LIN {X -0.184, Y -19.690, Z 18.700} C_DIS
   LIN {X 0.095, Y -20.163, Z 18.700} C_DIS
   LIN {X 0.765, Y -21.484, Z 18.700} C_DIS
   LIN {X 0.956, Y -22.494, Z 18.700} C_DIS
   LIN {X 0.778, Y -24.107, Z 18.700} C_DIS
   LIN {X 0.768, Y -24.353, Z 18.700} C_DIS
   LIN {X 0.683, Y -24.523, Z 18.700} C_DIS
   LIN {X 0.039, Y -25.176, Z 18.700} C_DIS
   LIN {X -1.565, Y -27.106, Z 18.700} C_DIS
   LIN {X -2.023, Y -27.501, Z 18.700} C_DIS
   LIN {X -2.702, Y -27.685, Z 18.700} C_DIS
   LIN {X -4.263, Y -27.893, Z 18.700} C_DIS
   LIN {X -4.894, Y -27.845, Z 18.700} C_DIS
   LIN {X -5.662, Y -27.602, Z 18.700} C_DIS
   LIN {X -6.185, Y -27.453, Z 18.700} C_DIS
   LIN {X -6.544, Y -27.180, Z 18.700}
   LaserEnd_Ext()
   LIN {X 0.074, Y 42.514, Z 18.700}
   LaserStart_Ext()
   LIN {X -0.388, Y 42.343, Z 18.700} C_DIS
   LIN {X -2.614, Y 41.518, Z 18.700} C_DIS
   LIN {X -3.480, Y 40.431, Z 18.700} C_DIS
   LIN {X -3.666, Y 39.839, Z 18.700} C_DIS
   LIN {X -3.933, Y 38.968, Z 18.700} C_DIS
   LIN {X -3.877, Y 38.326, Z 18.700} C_DIS
   LIN {X -3.817, Y 37.522, Z 18.700} C_DIS
   LIN {X -3.553, Y 36.446, Z 18.700} C_DIS
   LIN {X -3.518, Y 36.307, Z 18.700} C_DIS
   LIN {X -3.492, Y 36.196, Z 18.700} C_DIS
   LIN {X -3.157, Y 34.747, Z 18.700} C_DIS
   LIN {X -2.764, Y 32.822, Z 18.700} C_DIS
   LIN {X -2.683, Y 32.424, Z 18.700} C_DIS
   LIN {X -2.583, Y 31.822, Z 18.700} C_DIS
   LIN {X -2.259, Y 29.905, Z 18.700} C_DIS
   LIN {X -2.174, Y 29.276, Z 18.700} C_DIS
   LIN {X -2.026, Y 28.170, Z 18.700} C_DIS
   LIN {X -1.804, Y 26.224, Z 18.700} C_DIS
   LIN {X -1.527, Y 21.880, Z 18.700} C_DIS
   LIN {X -1.462, Y 20.734, Z 18.700} C_DIS
   LIN {X -1.462, Y 19.942, Z 18.700} C_DIS
   LIN {X -1.534, Y 15.412, Z 18.700} C_DIS
   LIN {X -1.749, Y 12.450, Z 18.700} C_DIS
   LIN {X -1.755, Y 12.285, Z 18.700} C_DIS
   LIN {X -1.795, Y 11.801, Z 18.700} C_DIS
   LIN {X -2.174, Y 8.729, Z 18.700} C_DIS
   LIN {X -2.302, Y 7.850, Z 18.700} C_DIS
   LIN {X -2.755, Y 5.576, Z 18.700} C_DIS
   LIN {X -3.323, Y 2.576, Z 18.700} C_DIS
   LIN {X -3.541, Y 1.648, Z 18.700} C_DIS
   LIN {X -5.722, Y -5.572, Z 18.700} C_DIS
   LIN {X -5.770, Y -5.725, Z 18.700} C_DIS
   LIN {X -5.824, Y -5.860, Z 18.700} C_DIS
   LIN {X -7.511, Y -10.111, Z 18.700} C_DIS
   LIN {X -8.322, Y -11.837, Z 18.700} C_DIS
   LIN {X -9.632, Y -14.546, Z 18.700} C_DIS
   LIN {X -9.994, Y -15.230, Z 18.700} C_DIS
   LIN {X -11.132, Y -17.238, Z 18.700} C_DIS
   LIN {X -11.749, Y -18.344, Z 18.700} C_DIS
   LIN {X -12.022, Y -19.074, Z 18.700} C_DIS
   LIN {X -12.873, Y -21.308, Z 18.700} C_DIS
   LIN {X -12.802, Y -24.694, Z 18.700} C_DIS
   LIN {X -12.798, Y -25.019, Z 18.700} C_DIS
   LIN {X -12.743, Y -25.160, Z 18.700} C_DIS
   LIN {X -12.472, Y -25.804, Z 18.700} C_DIS
   LIN {X -11.655, Y -27.758, Z 18.700} C_DIS
   LIN {X -10.921, Y -28.587, Z 18.700} C_DIS
   LIN {X -9.889, Y -29.793, Z 18.700} C_DIS
   LIN {X -8.777, Y -30.514, Z 18.700} C_DIS
   LIN {X -7.630, Y -31.202, Z 18.700} C_DIS
   LIN {X -6.964, Y -31.390, Z 18.700} C_DIS
   LIN {X -5.127, Y -31.859, Z 18.700} C_DIS
   LIN {X -2.530, Y -31.794, Z 18.700} C_DIS
   LIN {X -2.407, Y -31.779, Z 18.700} C_DIS
   LIN {X -2.291, Y -31.728, Z 18.700} C_DIS
   LIN {X 1.037, Y -30.354, Z 18.700} C_DIS
   LIN {X 2.203, Y -29.260, Z 18.700} C_DIS
   LIN {X 3.220, Y -28.251, Z 18.700} C_DIS
   LIN {X 4.167, Y -26.340, Z 18.700} C_DIS
   LIN {X 4.631, Y -25.432, Z 18.700} C_DIS
   LIN {X 4.832, Y -24.724, Z 18.700} C_DIS
   LIN {X 5.507, Y -22.287, Z 18.700} C_DIS
   LIN {X 6.244, Y -19.312, Z 18.700} C_DIS
   LIN {X 6.296, Y -19.100, Z 18.700} C_DIS
   LIN {X 6.353, Y -18.826, Z 18.700} C_DIS
   LIN {X 7.032, Y -15.668, Z 18.700} C_DIS
   LIN {X 7.452, Y -13.374, Z 18.700} C_DIS
   LIN {X 7.904, Y -10.693, Z 18.700} C_DIS
   LIN {X 8.410, Y -6.804, Z 18.700} C_DIS
   LIN {X 8.601, Y -5.119, Z 18.700} C_DIS
   LIN {X 8.928, Y -1.168, Z 18.700} C_DIS
   LIN {X 8.983, Y 0.851, Z 18.700} C_DIS
   LIN {X 9.138, Y 6.966, Z 18.700} C_DIS
   LIN {X 9.136, Y 7.901, Z 18.700} C_DIS
   LIN {X 9.053, Y 10.031, Z 18.700} C_DIS
   LIN {X 8.957, Y 12.408, Z 18.700} C_DIS
   LIN {X 8.769, Y 14.715, Z 18.700} C_DIS
   LIN {X 8.614, Y 16.718, Z 18.700} C_DIS
   LIN {X 8.410, Y 18.528, Z 18.700} C_DIS
   LIN {X 8.236, Y 19.999, Z 18.700} C_DIS
   LIN {X 7.494, Y 24.645, Z 18.700} C_DIS
   LIN {X 7.227, Y 26.349, Z 18.700} C_DIS
   LIN {X 7.179, Y 26.606, Z 18.700} C_DIS
   LIN {X 7.055, Y 27.190, Z 18.700} C_DIS
   LIN {X 6.376, Y 30.443, Z 18.700} C_DIS
   LIN {X 5.730, Y 33.096, Z 18.700} C_DIS
   LIN {X 5.569, Y 33.746, Z 18.700} C_DIS
   LIN {X 4.887, Y 36.234, Z 18.700} C_DIS
   LIN {X 4.824, Y 36.463, Z 18.700} C_DIS
   LIN {X 4.278, Y 38.303, Z 18.700} C_DIS
   LIN {X 3.974, Y 39.275, Z 18.700} C_DIS
   LIN {X 3.833, Y 39.720, Z 18.700} C_DIS
   LIN {X 3.557, Y 40.230, Z 18.700} C_DIS
   LIN {X 3.133, Y 41.017, Z 18.700} C_DIS
   LIN {X 2.483, Y 41.539, Z 18.700} C_DIS
   LIN {X 1.772, Y 42.105, Z 18.700} C_DIS
   LIN {X 0.360, Y 42.444, Z 18.700} C_DIS
   LIN {X 0.074, Y 42.514, Z 18.700}
   LaserEnd_Ext()
   LIN {X 2.153, Y 40.522, Z 18.700}
   LaserStart_Ext()
   LIN {X -2.129, Y 40.522, Z 18.700}
   LaserEnd_Ext()
   LIN {X -2.717, Y 39.522, Z 18.700}
   LaserStart_Ext()
   LIN {X 2.803, Y 39.522, Z 18.700}
   LaserEnd_Ext()
   LIN {X 3.161, Y 38.522, Z 18.700}
   LaserStart_Ext()
   LIN {X -2.891, Y 38.522, Z 18.700}
   LaserEnd_Ext()
   LIN {X -2.788, Y 37.522, Z 18.700}
   LaserStart_Ext()
   LIN {X 3.467, Y 37.522, Z 18.700}
   LaserEnd_Ext()
   LIN {X 3.764, Y 36.522, Z 18.700}
   LaserStart_Ext()
   LIN {X -2.542, Y 36.522, Z 18.700}
   LaserEnd_Ext()
   LIN {X -2.310, Y 35.522, Z 18.700}
   LaserStart_Ext()
   LIN {X 4.045, Y 35.522, Z 18.700}
   LaserEnd_Ext()
   LIN {X 4.319, Y 34.522, Z 18.700}
   LaserStart_Ext()
   LIN {X -2.090, Y 34.522, Z 18.700}
   LaserEnd_Ext()
   LIN {X -1.886, Y 33.522, Z 18.700}
   LaserStart_Ext()
   LIN {X 4.593, Y 33.522, Z 18.700}
   LaserEnd_Ext()
   LIN {X 4.841, Y 32.522, Z 18.700}
   LaserStart_Ext()
   LIN {X -1.686, Y 32.522, Z 18.700}
   LaserEnd_Ext()
   LIN {X -1.518, Y 31.522, Z 18.700}
   LaserStart_Ext()
   LIN {X 5.084, Y 31.522, Z 18.700}
   LaserEnd_Ext()
   LIN {X 5.327, Y 30.522, Z 18.700}
   LaserStart_Ext()
   LIN {X -1.349, Y 30.522, Z 18.700}
   LaserEnd_Ext()
   LIN {X -1.198, Y 29.522, Z 18.700}
   LaserStart_Ext()
   LIN {X 5.547, Y 29.522, Z 18.700}
   LaserEnd_Ext()
   LIN {X 5.756, Y 28.522, Z 18.700}
   LaserStart_Ext()
   LIN {X -1.064, Y 28.522, Z 18.700}
   LaserEnd_Ext()
   LIN {X -0.946, Y 27.522, Z 18.700}
   LaserStart_Ext()
   LIN {X 5.964, Y 27.522, Z 18.700}
   LaserEnd_Ext()
   LIN {X 6.175, Y 26.522, Z 18.700}
   LaserStart_Ext()
   LIN {X -0.832, Y 26.522, Z 18.700}
   LaserEnd_Ext()
   LIN {X -0.757, Y 25.522, Z 18.700}
   LaserStart_Ext()
   LIN {X 6.345, Y 25.522, Z 18.700}
   LaserEnd_Ext()
   LIN {X 6.501, Y 24.522, Z 18.700}
   LaserStart_Ext()
   LIN {X -0.694, Y 24.522, Z 18.700}
   LaserEnd_Ext()
   LIN {X -0.630, Y 23.522, Z 18.700}
   LaserStart_Ext()
   LIN {X 6.661, Y 23.522, Z 18.700}
   LaserEnd_Ext()
   LIN {X 6.821, Y 22.522, Z 18.700}
   LaserStart_Ext()
   LIN {X -0.566, Y 22.522, Z 18.700}
   LaserEnd_Ext()
   LIN {X -0.505, Y 21.522, Z 18.700}
   LaserStart_Ext()
   LIN {X 6.980, Y 21.522, Z 18.700}
   LaserEnd_Ext()
   LIN {X 7.140, Y 20.522, Z 18.700}
   LaserStart_Ext()
   LIN {X -0.462, Y 20.522, Z 18.700}
   LaserEnd_Ext()
   LIN {X -0.468, Y 19.522, Z 18.700}
   LaserStart_Ext()
   LIN {X 7.286, Y 19.522, Z 18.700}
   LaserEnd_Ext()
   LIN {X 7.404, Y 18.522, Z 18.700}
   LaserStart_Ext()
   LIN {X -0.484, Y 18.522, Z 18.700}
   LaserEnd_Ext()
   LIN {X -0.500, Y 17.522, Z 18.700}
   LaserStart_Ext()
   LIN {X 7.517, Y 17.522, Z 18.700}
   LaserEnd_Ext()
   LIN {X 7.626, Y 16.522, Z 18.700}
   LaserStart_Ext()
   LIN {X -0.516, Y 16.522, Z 18.700}
   LaserEnd_Ext()
   LIN {X -0.532, Y 15.522, Z 18.700}
   LaserStart_Ext()
   LIN {X 7.704, Y 15.522, Z 18.700}
   LaserEnd_Ext()
   LIN {X 7.781, Y 14.522, Z 18.700}
   LaserStart_Ext()
   LIN {X -0.596, Y 14.522, Z 18.700}
   LaserEnd_Ext()
   LIN {X -0.668, Y 13.522, Z 18.700}
   LaserStart_Ext()
   LIN {X 7.863, Y 13.522, Z 18.700}
   LaserEnd_Ext()
   LIN {X 7.944, Y 12.522, Z 18.700}
   LaserStart_Ext()
   LIN {X -0.741, Y 12.522, Z 18.700}
   LaserEnd_Ext()
   LIN {X -0.822, Y 11.522, Z 18.700}
   LaserStart_Ext()
   LIN {X 7.992, Y 11.522, Z 18.700}
   LaserEnd_Ext()
   LIN {X 8.032, Y 10.522, Z 18.700}
   LaserStart_Ext()
   LIN {X -0.945, Y 10.522, Z 18.700}
   LaserEnd_Ext()
   LIN {X -1.069, Y 9.522, Z 18.700}
   LaserStart_Ext()
   LIN {X 8.072, Y 9.522, Z 18.700}
   LaserEnd_Ext()
   LIN {X 8.111, Y 8.522, Z 18.700}
   LaserStart_Ext()
   LIN {X -1.194, Y 8.522, Z 18.700}
   LaserEnd_Ext()
   LIN {X -1.348, Y 7.522, Z 18.700}
   LaserStart_Ext()
   LIN {X 8.137, Y 7.522, Z 18.700}
   LaserEnd_Ext()
   LIN {X 8.127, Y 6.522, Z 18.700}
   LaserStart_Ext()
   LIN {X -1.547, Y 6.522, Z 18.700}
   LaserEnd_Ext()
   LIN {X -1.746, Y 5.522, Z 18.700}
   LaserStart_Ext()
   LIN {X 8.101, Y 5.522, Z 18.700}
   LaserEnd_Ext()
   LIN {X 8.076, Y 4.522, Z 18.700}
   LaserStart_Ext()
   LIN {X -1.937, Y 4.522, Z 18.700}
   LaserEnd_Ext()
   LIN {X -2.126, Y 3.522, Z 18.700}
   LaserStart_Ext()
   LIN {X 8.050, Y 3.522, Z 18.700}
   LaserEnd_Ext()
   LIN {X 8.025, Y 2.522, Z 18.700}
   LaserStart_Ext()
   LIN {X -2.315, Y 2.522, Z 18.700}
   LaserEnd_Ext()
   LIN {X -2.544, Y 1.522, Z 18.700}
   LaserStart_Ext()
   LIN {X 7.999, Y 1.522, Z 18.700}
   LaserEnd_Ext()
   LIN {X 7.973, Y 0.522, Z 18.700}
   LaserStart_Ext()
   LIN {X -2.837, Y 0.522, Z 18.700}
   LaserEnd_Ext()
   LIN {X -3.139, Y -0.478, Z 18.700}
   LaserStart_Ext()
   LIN {X 7.946, Y -0.478, Z 18.700}
   LaserEnd_Ext()
   LIN {X 7.899, Y -1.478, Z 18.700}
   LaserStart_Ext()
   LIN {X -3.441, Y -1.478, Z 18.700}
   LaserEnd_Ext()
   LIN {X -3.743, Y -2.478, Z 18.700}
   LaserStart_Ext()
   LIN {X 7.816, Y -2.478, Z 18.700}
   LaserEnd_Ext()
   LIN {X 7.733, Y -3.478, Z 18.700}
   LaserStart_Ext()
   LIN {X -4.045, Y -3.478, Z 18.700}
   LaserEnd_Ext()
   LIN {X -4.347, Y -4.478, Z 18.700}
   LaserStart_Ext()
   LIN {X 7.651, Y -4.478, Z 18.700}
   LaserEnd_Ext()
   LIN {X 7.554, Y -5.478, Z 18.700}
   LaserStart_Ext()
   LIN {X -4.649, Y -5.478, Z 18.700}
   LaserEnd_Ext()
   LIN {X -4.993, Y -6.478, Z 18.700}
   LaserStart_Ext()
   LIN {X 7.440, Y -6.478, Z 18.700}
   LaserEnd_Ext()
   LIN {X 7.314, Y -7.478, Z 18.700}
   LaserStart_Ext()
   LIN {X -5.390, Y -7.478, Z 18.700}
   LaserEnd_Ext()
   LIN {X -5.787, Y -8.478, Z 18.700}
   LaserStart_Ext()
   LIN {X 7.184, Y -8.478, Z 18.700}
   LaserEnd_Ext()
   LIN {X 7.053, Y -9.478, Z 18.700}
   LaserStart_Ext()
   LIN {X -6.184, Y -9.478, Z 18.700}
   LaserEnd_Ext()
   LIN {X -6.581, Y -10.478, Z 18.700}
   LaserStart_Ext()
   LIN {X 6.923, Y -10.478, Z 18.700}
   LaserEnd_Ext()
   LIN {X 6.757, Y -11.478, Z 18.700}
   LaserStart_Ext()
   LIN {X -7.049, Y -11.478, Z 18.700}
   LaserEnd_Ext()
   LIN {X -7.521, Y -12.478, Z 18.700}
   LaserStart_Ext()
   LIN {X 6.589, Y -12.478, Z 18.700}
   LaserEnd_Ext()
   LIN {X 6.416, Y -13.478, Z 18.700}
   LaserStart_Ext()
   LIN {X -8.005, Y -13.478, Z 18.700}
   LaserEnd_Ext()
   LIN {X -8.488, Y -14.478, Z 18.700}
   LaserStart_Ext()
   LIN {X 6.233, Y -14.478, Z 18.700}
   LaserEnd_Ext()
   LIN {X 6.050, Y -15.478, Z 18.700}
   LaserStart_Ext()
   LIN {X -8.994, Y -15.478, Z 18.700}
   LaserEnd_Ext()
   LIN {X -9.552, Y -16.478, Z 18.700}
   LaserStart_Ext()
   LIN {X 5.835, Y -16.478, Z 18.700}
   LaserEnd_Ext()
   LIN {X 5.620, Y -17.478, Z 18.700}
   LaserStart_Ext()
   LIN {X -1.462, Y -17.478, Z 18.700}
   LaserEnd_Ext()
   LIN {X -6.497, Y -17.478, Z 18.700}
   LaserStart_Ext()
   LIN {X -10.119, Y -17.478, Z 18.700}
   LaserEnd_Ext()
   LIN {X -10.679, Y -18.478, Z 18.700}
   LaserStart_Ext()
   LIN {X -7.803, Y -18.478, Z 18.700}
   LaserEnd_Ext()
   LIN {X -0.116, Y -18.478, Z 18.700}
   LaserStart_Ext()
   LIN {X 5.405, Y -18.478, Z 18.700}
   LaserEnd_Ext()
   LIN {X 5.173, Y -19.478, Z 18.700}
   LaserStart_Ext()
   LIN {X 0.852, Y -19.478, Z 18.700}
   LaserEnd_Ext()
   LIN {X -8.904, Y -19.478, Z 18.700}
   LaserStart_Ext()
   LIN {X -11.106, Y -19.478, Z 18.700}
   LaserEnd_Ext()
   LIN {X -11.487, Y -20.478, Z 18.700}
   LaserStart_Ext()
   LIN {X -9.378, Y -20.478, Z 18.700}
   LaserEnd_Ext()
   LIN {X 1.376, Y -20.478, Z 18.700}
   LaserStart_Ext()
   LIN {X 4.925, Y -20.478, Z 18.700}
   LaserEnd_Ext()
   LIN {X 4.677, Y -21.478, Z 18.700}
   LaserStart_Ext()
   LIN {X 1.781, Y -21.478, Z 18.700}
   LaserEnd_Ext()
   LIN {X -9.805, Y -21.478, Z 18.700}
   LaserStart_Ext()
   LIN {X -11.868, Y -21.478, Z 18.700}
   LaserEnd_Ext()
   LIN {X -11.849, Y -22.478, Z 18.700}
   LaserStart_Ext()
   LIN {X -9.961, Y -22.478, Z 18.700}
   LaserEnd_Ext()
   LIN {X 1.955, Y -22.478, Z 18.700}
   LaserStart_Ext()
   LIN {X 4.416, Y -22.478, Z 18.700}
   LaserEnd_Ext()
   LIN {X 4.139, Y -23.478, Z 18.700}
   LaserStart_Ext()
   LIN {X 1.853, Y -23.478, Z 18.700}
   LaserEnd_Ext()
   LIN {X -9.983, Y -23.478, Z 18.700}
   LaserStart_Ext()
   LIN {X -11.828, Y -23.478, Z 18.700}
   LaserEnd_Ext()
   LIN {X -11.807, Y -24.478, Z 18.700}
   LaserStart_Ext()
   LIN {X -9.759, Y -24.478, Z 18.700}
   LaserEnd_Ext()
   LIN {X 1.759, Y -24.478, Z 18.700}
   LaserStart_Ext()
   LIN {X 3.862, Y -24.478, Z 18.700}
   LaserEnd_Ext()
   LIN {X 3.484, Y -25.478, Z 18.700}
   LaserStart_Ext()
   LIN {X 1.145, Y -25.478, Z 18.700}
   LaserEnd_Ext()
   LIN {X -9.414, Y -25.478, Z 18.700}
   LaserStart_Ext()
   LIN {X -11.524, Y -25.478, Z 18.700}
   LaserEnd_Ext()
   LIN {X -11.106, Y -26.478, Z 18.700}
   LaserStart_Ext()
   LIN {X -8.816, Y -26.478, Z 18.700}
   LaserEnd_Ext()
   LIN {X 0.257, Y -26.478, Z 18.700}
   LaserStart_Ext()
   LIN {X 2.983, Y -26.478, Z 18.700}
   LaserEnd_Ext()
   LIN {X 2.487, Y -27.478, Z 18.700}
   LaserStart_Ext()
   LIN {X -0.574, Y -27.478, Z 18.700}
   LaserEnd_Ext()
   LIN {X -7.707, Y -27.478, Z 18.700}
   LaserStart_Ext()
   LIN {X -10.567, Y -27.478, Z 18.700}
   LaserEnd_Ext()
   LIN {X -9.698, Y -28.478, Z 18.700}
   LaserStart_Ext()
   LIN {X -6.237, Y -28.478, Z 18.700}
   LaserEnd_Ext()
   LIN {X -1.807, Y -28.478, Z 18.700}
   LaserStart_Ext()
   LIN {X 1.572, Y -28.478, Z 18.700}
   LaserEnd_Ext()
   LIN {X 0.509, Y -29.478, Z 18.700}
   LaserStart_Ext()
   LIN {X -8.536, Y -29.478, Z 18.700}
   LaserEnd_Ext()
   LIN {X -6.493, Y -30.478, Z 18.700}
   LaserStart_Ext()
   LIN {X -1.885, Y -30.478, Z 18.700}
   LaserEnd_Ext()
   LIN {X -6.100, Y -27.413, Z 19.550}
   LaserStart_Ext()
   LIN {X -7.561, Y -26.301, Z 19.550} C_DIS
   LIN {X -7.793, Y -26.092, Z 19.550} C_DIS
   LIN {X -8.501, Y -24.912, Z 19.550} C_DIS
   LIN {X -8.813, Y -24.007, Z 19.550} C_DIS
   LIN {X -8.928, Y -23.216, Z 19.550} C_DIS
   LIN {X -8.912, Y -22.461, Z 19.550} C_DIS
   LIN {X -8.614, Y -21.240, Z 19.550} C_DIS
   LIN {X -8.238, Y -20.363, Z 19.550} C_DIS
   LIN {X -7.705, Y -19.610, Z 19.550} C_DIS
   LIN {X -7.006, Y -19.067, Z 19.550} C_DIS
   LIN {X -5.907, Y -18.286, Z 19.550} C_DIS
   LIN {X -4.103, Y -17.923, Z 19.550} C_DIS
   LIN {X -3.878, Y -17.878, Z 19.550} C_DIS
   LIN {X -3.692, Y -17.920, Z 19.550} C_DIS
   LIN {X -1.802, Y -18.341, Z 19.550} C_DIS
   LIN {X -0.204, Y -19.569, Z 19.550} C_DIS
   LIN {X -0.117, Y -19.635, Z 19.550} C_DIS
   LIN {X -0.056, Y -19.762, Z 19.550} C_DIS
   LIN {X 0.896, Y -21.639, Z 19.550} C_DIS
   LIN {X 1.006, Y -22.224, Z 19.550} C_DIS
   LIN {X 0.903, Y -23.157, Z 19.550} C_DIS
   LIN {X 0.859, Y -24.247, Z 19.550} C_DIS
   LIN {X 0.481, Y -25.003, Z 19.550} C_DIS
   LIN {X -1.844, Y -27.359, Z 19.550} C_DIS
   LIN {X -1.994, Y -27.476, Z 19.550} C_DIS
   LIN {X -2.142, Y -27.505, Z 19.550} C_DIS
   LIN {X -4.502, Y -27.849, Z 19.550} C_DIS
   LIN {X -5.043, Y -27.714, Z 19.550} C_DIS
   LIN {X -6.100, Y -27.413, Z 19.550}
   LaserEnd_Ext()
   LIN {X -11.686, Y -18.315, Z 19.550}
   LaserStart_Ext()
   LIN {X -12.363, Y -20.122, Z 19.550} C_DIS
   LIN {X -12.805, Y -21.282, Z 19.550} C_DIS
   LIN {X -12.759, Y -23.477, Z 19.550} C_DIS
   LIN {X -12.720, Y -24.992, Z 19.550} C_DIS
   LIN {X -12.388, Y -25.778, Z 19.550} C_DIS
   LIN {X -11.574, Y -27.726, Z 19.550} C_DIS
   LIN {X -9.684, Y -29.860, Z 19.550} C_DIS
   LIN {X -7.476, Y -31.189, Z 19.550} C_DIS
   LIN {X -6.204, Y -31.549, Z 19.550} C_DIS
   LIN {X -5.254, Y -31.792, Z 19.550} C_DIS
   LIN {X -3.751, Y -31.754, Z 19.550} C_DIS
   LIN {X -2.424, Y -31.751, Z 19.550} C_DIS
   LIN {X -0.109, Y -30.793, Z 19.550} C_DIS
   LIN {X 1.177, Y -30.262, Z 19.550} C_DIS
   LIN {X 1.568, Y -29.896, Z 19.550} C_DIS
   LIN {X 3.348, Y -28.128, Z 19.550} C_DIS
   LIN {X 4.497, Y -25.809, Z 19.550} C_DIS
   LIN {X 4.709, Y -25.365, Z 19.550} C_DIS
   LIN {X 4.970, Y -24.413, Z 19.550} C_DIS
   LIN {X 5.578, Y -22.219, Z 19.550} C_DIS
   LIN {X 5.927, Y -20.808, Z 19.550} C_DIS
   LIN {X 6.348, Y -19.082, Z 19.550} C_DIS
   LIN {X 6.814, Y -16.862, Z 19.550} C_DIS
   LIN {X 7.117, Y -15.455, Z 19.550} C_DIS
   LIN {X 7.304, Y -14.433, Z 19.550} C_DIS
   LIN {X 7.964, Y -10.519, Z 19.550} C_DIS
   LIN {X 8.268, Y -8.183, Z 19.550} C_DIS
   LIN {X 8.669, Y -4.642, Z 19.550} C_DIS
   LIN {X 8.896, Y -1.901, Z 19.550} C_DIS
   LIN {X 9.087, Y 5.130, Z 19.550} C_DIS
   LIN {X 9.144, Y 7.345, Z 19.550} C_DIS
   LIN {X 9.143, Y 7.684, Z 19.550} C_DIS
   LIN {X 9.113, Y 8.456, Z 19.550} C_DIS
   LIN {X 8.951, Y 12.449, Z 19.550} C_DIS
   LIN {X 8.636, Y 16.325, Z 19.550} C_DIS
   LIN {X 8.612, Y 16.628, Z 19.550} C_DIS
   LIN {X 8.581, Y 16.901, Z 19.550} C_DIS
   LIN {X 8.190, Y 20.223, Z 19.550} C_DIS
   LIN {X 7.378, Y 25.302, Z 19.550} C_DIS
   LIN {X 7.182, Y 26.451, Z 19.550} C_DIS
   LIN {X 6.968, Y 27.455, Z 19.550} C_DIS
   LIN {X 6.364, Y 30.348, Z 19.550} C_DIS
   LIN {X 5.945, Y 32.070, Z 19.550} C_DIS
   LIN {X 5.524, Y 33.763, Z 19.550} C_DIS
   LIN {X 5.284, Y 34.641, Z 19.550} C_DIS
   LIN {X 4.789, Y 36.430, Z 19.550} C_DIS
   LIN {X 4.288, Y 38.106, Z 19.550} C_DIS
   LIN {X 4.211, Y 38.362, Z 19.550} C_DIS
   LIN {X 4.118, Y 38.654, Z 19.550} C_DIS
   LIN {X 3.761, Y 39.784, Z 19.550} C_DIS
   LIN {X 3.326, Y 40.589, Z 19.550} C_DIS
   LIN {X 3.059, Y 41.079, Z 19.550} C_DIS
   LIN {X 2.382, Y 41.616, Z 19.550} C_DIS
   LIN {X 1.695, Y 42.164, Z 19.550} C_DIS
   LIN {X 1.139, Y 42.298, Z 19.550} C_DIS
   LIN {X -0.004, Y 42.569, Z 19.550} C_DIS
   LIN {X -1.763, Y 41.910, Z 19.550} C_DIS
   LIN {X -2.689, Y 41.567, Z 19.550} C_DIS
   LIN {X -3.056, Y 41.107, Z 19.550} C_DIS
   LIN {X -3.568, Y 40.449, Z 19.550} C_DIS
   LIN {X -3.770, Y 39.733, Z 19.550} C_DIS
   LIN {X -4.008, Y 38.956, Z 19.550} C_DIS
   LIN {X -3.929, Y 38.038, Z 19.550} C_DIS
   LIN {X -3.884, Y 37.568, Z 19.550} C_DIS
   LIN {X -3.794, Y 37.210, Z 19.550} C_DIS
   LIN {X -3.582, Y 36.353, Z 19.550} C_DIS
   LIN {X -3.244, Y 34.916, Z 19.550} C_DIS
   LIN {X -3.216, Y 34.795, Z 19.550} C_DIS
   LIN {X -3.169, Y 34.564, Z 19.550} C_DIS
   LIN {X -2.738, Y 32.472, Z 19.550} C_DIS
   LIN {X -2.450, Y 30.812, Z 19.550} C_DIS
   LIN {X -2.328, Y 30.089, Z 19.550} C_DIS
   LIN {X -2.096, Y 28.382, Z 19.550} C_DIS
   LIN {X -2.000, Y 27.662, Z 19.550} C_DIS
   LIN {X -1.856, Y 26.395, Z 19.550} C_DIS
   LIN {X -1.494, Y 20.713, Z 19.550} C_DIS
   LIN {X -1.483, Y 20.520, Z 19.550} C_DIS
   LIN {X -1.483, Y 20.386, Z 19.550} C_DIS
   LIN {X -1.566, Y 15.103, Z 19.550} C_DIS
   LIN {X -1.804, Y 11.836, Z 19.550} C_DIS
   LIN {X -1.818, Y 11.701, Z 19.550} C_DIS
   LIN {X -2.197, Y 8.637, Z 19.550} C_DIS
   LIN {X -2.259, Y 8.139, Z 19.550} C_DIS
   LIN {X -2.278, Y 8.035, Z 19.550} C_DIS
   LIN {X -3.263, Y 2.832, Z 19.550} C_DIS
   LIN {X -3.642, Y 1.223, Z 19.550} C_DIS
   LIN {X -5.286, Y -4.220, Z 19.550} C_DIS
   LIN {X -5.789, Y -5.833, Z 19.550} C_DIS
   LIN {X -6.357, Y -7.255, Z 19.550} C_DIS
   LIN {X -7.545, Y -10.249, Z 19.550} C_DIS
   LIN {X -8.117, Y -11.465, Z 19.550} C_DIS
   LIN {X -9.743, Y -14.830, Z 19.550} C_DIS
   LIN {X -9.844, Y -15.021, Z 19.550} C_DIS
   LIN {X -10.161, Y -15.579, Z 19.550} C_DIS
   LIN {X -11.686, Y -18.315, Z 19.550}
   LaserEnd_Ext()
   LIN {X -11.280, Y -25.836, Z 19.550}
   LaserStart_Ext()
   LIN {X -11.280, Y -20.081, Z 19.550}
   LaserEnd_Ext()
   LIN {X -10.280, Y -17.847, Z 19.550}
   LaserStart_Ext()
   LIN {X -10.280, Y -27.679, Z 19.550}
   LaserEnd_Ext()
   LIN {X -9.280, Y -28.808, Z 19.550}
   LaserStart_Ext()
   LIN {X -9.280, Y -25.557, Z 19.550}
   LaserEnd_Ext()
   LIN {X -9.280, Y -20.255, Z 19.550}
   LaserStart_Ext()
   LIN {X -9.280, Y -16.053, Z 19.550}
   LaserEnd_Ext()
   LIN {X -8.280, Y -14.101, Z 19.550}
   LaserStart_Ext()
   LIN {X -8.280, Y -18.790, Z 19.550}
   LaserEnd_Ext()
   LIN {X -8.280, Y -26.999, Z 19.550}
   LaserStart_Ext()
   LIN {X -8.280, Y -29.541, Z 19.550}
   LaserEnd_Ext()
   LIN {X -7.280, Y -30.141, Z 19.550}
   LaserStart_Ext()
   LIN {X -7.280, Y -27.771, Z 19.550}
   LaserEnd_Ext()
   LIN {X -7.280, Y -18.035, Z 19.550}
   LaserStart_Ext()
   LIN {X -7.280, Y -12.032, Z 19.550}
   LaserEnd_Ext()
   LIN {X -6.280, Y -9.772, Z 19.550}
   LaserStart_Ext()
   LIN {X -6.280, Y -17.359, Z 19.550}
   LaserEnd_Ext()
   LIN {X -6.280, Y -28.401, Z 19.550}
   LaserStart_Ext()
   LIN {X -6.280, Y -30.488, Z 19.550}
   LaserEnd_Ext()
   LIN {X -5.280, Y -30.753, Z 19.550}
   LaserStart_Ext()
   LIN {X -5.280, Y -28.685, Z 19.550}
   LaserEnd_Ext()
   LIN {X -5.280, Y -17.140, Z 19.550}
   LaserStart_Ext()
   LIN {X -5.280, Y -7.255, Z 19.550}
   LaserEnd_Ext()
   LIN {X -4.280, Y -4.347, Z 19.550}
   LaserStart_Ext()
   LIN {X -4.280, Y -16.938, Z 19.550}
   LaserEnd_Ext()
   LIN {X -4.280, Y -28.827, Z 19.550}
   LaserStart_Ext()
   LIN {X -4.280, Y -30.767, Z 19.550}
   LaserEnd_Ext()
   LIN {X -3.280, Y -30.753, Z 19.550}
   LaserStart_Ext()
   LIN {X -3.280, Y -28.682, Z 19.550}
   LaserEnd_Ext()
   LIN {X -3.280, Y -16.988, Z 19.550}
   LaserStart_Ext()
   LIN {X -3.280, Y -1.036, Z 19.550}
   LaserEnd_Ext()
   LIN {X -2.280, Y 40.476, Z 19.550}
   LaserStart_Ext()
   LIN {X -2.280, Y 35.183, Z 19.550}
   LaserEnd_Ext()
   LIN {X -2.280, Y 2.649, Z 19.550}
   LaserStart_Ext()
   LIN {X -2.280, Y -17.210, Z 19.550}
   LaserEnd_Ext()
   LIN {X -2.280, Y -28.536, Z 19.550}
   LaserStart_Ext()
   LIN {X -2.280, Y -30.609, Z 19.550}
   LaserEnd_Ext()
   LIN {X -1.280, Y -30.195, Z 19.550}
   LaserStart_Ext()
   LIN {X -1.280, Y -28.187, Z 19.550}
   LaserEnd_Ext()
   LIN {X -1.280, Y -17.488, Z 19.550}
   LaserStart_Ext()
   LIN {X -1.280, Y 7.929, Z 19.550}
   LaserEnd_Ext()
   LIN {X -1.280, Y 29.800, Z 19.550}
   LaserStart_Ext()
   LIN {X -1.280, Y 41.024, Z 19.550}
   LaserEnd_Ext()
   LIN {X -0.280, Y 41.398, Z 19.550}
   LaserStart_Ext()
   LIN {X -0.280, Y -18.249, Z 19.550}
   LaserEnd_Ext()
   LIN {X -0.280, Y -27.198, Z 19.550}
   LaserStart_Ext()
   LIN {X -0.280, Y -29.781, Z 19.550}
   LaserEnd_Ext()
   LIN {X 0.720, Y -29.320, Z 19.550}
   LaserStart_Ext()
   LIN {X 0.720, Y -26.184, Z 19.550}
   LaserEnd_Ext()
   LIN {X 0.720, Y -19.090, Z 19.550}
   LaserStart_Ext()
   LIN {X 0.720, Y 41.369, Z 19.550}
   LaserEnd_Ext()
   LIN {X 1.720, Y 40.865, Z 19.550}
   LaserStart_Ext()
   LIN {X 1.720, Y -21.054, Z 19.550}
   LaserEnd_Ext()
   LIN {X 1.720, Y -24.761, Z 19.550}
   LaserStart_Ext()
   LIN {X 1.720, Y -28.335, Z 19.550}
   LaserEnd_Ext()
   LIN {X 2.720, Y -27.143, Z 19.550}
   LaserStart_Ext()
   LIN {X 2.720, Y 39.607, Z 19.550}
   LaserEnd_Ext()
   LIN {X 3.720, Y 36.515, Z 19.550}
   LaserStart_Ext()
   LIN {X 3.720, Y -25.116, Z 19.550}
   LaserEnd_Ext()
   LIN {X 4.720, Y -21.521, Z 19.550}
   LaserStart_Ext()
   LIN {X 4.720, Y 32.852, Z 19.550}
   LaserEnd_Ext()
   LIN {X 5.720, Y 28.539, Z 19.550}
   LaserStart_Ext()
   LIN {X 5.720, Y -17.207, Z 19.550}
   LaserEnd_Ext()
   LIN {X 6.720, Y -11.880, Z 19.550}
   LaserStart_Ext()
   LIN {X 6.720, Y 23.083, Z 19.550}
   LaserEnd_Ext()
   LIN {X 7.720, Y 15.245, Z 19.550}
   LaserStart_Ext()
   LIN {X 7.720, Y -3.987, Z 19.550}
   LaserEnd_Ext()
   LIN {X -1.224, Y -18.685, Z 20.400}
   LaserStart_Ext()
   LIN {X -0.050, Y -19.580, Z 20.400} C_DIS
   LIN {X 0.768, Y -21.285, Z 20.400} C_DIS
   LIN {X 1.027, Y -21.795, Z 20.400} C_DIS
   LIN {X 1.056, Y -21.954, Z 20.400} C_DIS
   LIN {X 1.029, Y -22.207, Z 20.400} C_DIS
   LIN {X 0.950, Y -24.142, Z 20.400} C_DIS
   LIN {X 0.279, Y -25.483, Z 20.400} C_DIS
   LIN {X -0.760, Y -26.536, Z 20.400} C_DIS
   LIN {X -1.897, Y -27.420, Z 20.400} C_DIS
   LIN {X -3.019, Y -27.645, Z 20.400} C_DIS
   LIN {X -4.209, Y -27.818, Z 20.400} C_DIS
   LIN {X -5.783, Y -27.424, Z 20.400} C_DIS
   LIN {X -6.015, Y -27.372, Z 20.400} C_DIS
   LIN {X -6.161, Y -27.262, Z 20.400} C_DIS
   LIN {X -7.660, Y -26.125, Z 20.400} C_DIS
   LIN {X -8.379, Y -24.855, Z 20.400} C_DIS
   LIN {X -8.592, Y -24.501, Z 20.400} C_DIS
   LIN {X -8.666, Y -24.287, Z 20.400} C_DIS
   LIN {X -8.872, Y -22.871, Z 20.400} C_DIS
   LIN {X -8.869, Y -22.747, Z 20.400} C_DIS
   LIN {X -8.357, Y -20.646, Z 20.400} C_DIS
   LIN {X -8.243, Y -20.465, Z 20.400} C_DIS
   LIN {X -7.534, Y -19.449, Z 20.400} C_DIS
   LIN {X -6.941, Y -19.026, Z 20.400} C_DIS
   LIN {X -5.843, Y -18.245, Z 20.400} C_DIS
   LIN {X -3.797, Y -17.832, Z 20.400} C_DIS
   LIN {X -1.738, Y -18.290, Z 20.400} C_DIS
   LIN {X -1.224, Y -18.685, Z 20.400}
   LaserEnd_Ext()
   LIN {X 4.788, Y -25.298, Z 20.400}
   LaserStart_Ext()
   LIN {X 5.618, Y -22.265, Z 20.400} C_DIS
   LIN {X 5.649, Y -22.150, Z 20.400} C_DIS
   LIN {X 5.681, Y -22.014, Z 20.400} C_DIS
   LIN {X 6.401, Y -19.065, Z 20.400} C_DIS
   LIN {X 7.126, Y -15.611, Z 20.400} C_DIS
   LIN {X 7.195, Y -15.274, Z 20.400} C_DIS
   LIN {X 7.428, Y -13.875, Z 20.400} C_DIS
   LIN {X 8.024, Y -10.345, Z 20.400} C_DIS
   LIN {X 8.126, Y -9.561, Z 20.400} C_DIS
   LIN {X 8.738, Y -4.166, Z 20.400} C_DIS
   LIN {X 8.864, Y -2.635, Z 20.400} C_DIS
   LIN {X 9.065, Y 4.731, Z 20.400} C_DIS
   LIN {X 9.150, Y 7.181, Z 20.400} C_DIS
   LIN {X 9.131, Y 7.901, Z 20.400} C_DIS
   LIN {X 8.945, Y 12.490, Z 20.400} C_DIS
   LIN {X 8.647, Y 16.155, Z 20.400} C_DIS
   LIN {X 8.440, Y 17.926, Z 20.400} C_DIS
   LIN {X 8.143, Y 20.446, Z 20.400} C_DIS
   LIN {X 7.618, Y 23.732, Z 20.400} C_DIS
   LIN {X 7.144, Y 26.505, Z 20.400} C_DIS
   LIN {X 6.629, Y 28.925, Z 20.400} C_DIS
   LIN {X 6.352, Y 30.253, Z 20.400} C_DIS
   LIN {X 6.159, Y 31.043, Z 20.400} C_DIS
   LIN {X 5.834, Y 32.354, Z 20.400} C_DIS
   LIN {X 5.480, Y 33.781, Z 20.400} C_DIS
   LIN {X 4.940, Y 35.725, Z 20.400} C_DIS
   LIN {X 4.756, Y 36.390, Z 20.400} C_DIS
   LIN {X 4.678, Y 36.652, Z 20.400} C_DIS
   LIN {X 4.154, Y 38.390, Z 20.400} C_DIS
   LIN {X 3.813, Y 39.461, Z 20.400} C_DIS
   LIN {X 3.689, Y 39.849, Z 20.400} C_DIS
   LIN {X 3.455, Y 40.275, Z 20.400} C_DIS
   LIN {X 2.984, Y 41.141, Z 20.400} C_DIS
   LIN {X 2.264, Y 41.712, Z 20.400} C_DIS
   LIN {X 1.618, Y 42.223, Z 20.400} C_DIS
   LIN {X 0.339, Y 42.523, Z 20.400} C_DIS
   LIN {X -0.083, Y 42.623, Z 20.400} C_DIS
   LIN {X -0.778, Y 42.363, Z 20.400} C_DIS
   LIN {X -2.705, Y 41.666, Z 20.400} C_DIS
   LIN {X -3.364, Y 40.832, Z 20.400} C_DIS
   LIN {X -3.671, Y 40.438, Z 20.400} C_DIS
   LIN {X -3.866, Y 39.746, Z 20.400} C_DIS
   LIN {X -4.079, Y 38.991, Z 20.400} C_DIS
   LIN {X -4.033, Y 38.475, Z 20.400} C_DIS
   LIN {X -3.950, Y 37.613, Z 20.400} C_DIS
   LIN {X -3.705, Y 36.636, Z 20.400} C_DIS
   LIN {X -3.645, Y 36.400, Z 20.400} C_DIS
   LIN {X -3.600, Y 36.212, Z 20.400} C_DIS
   LIN {X -3.276, Y 34.842, Z 20.400} C_DIS
   LIN {X -2.847, Y 32.784, Z 20.400} C_DIS
   LIN {X -2.792, Y 32.520, Z 20.400} C_DIS
   LIN {X -2.732, Y 32.171, Z 20.400} C_DIS
   LIN {X -2.384, Y 30.184, Z 20.400} C_DIS
   LIN {X -2.178, Y 28.659, Z 20.400} C_DIS
   LIN {X -2.019, Y 27.488, Z 20.400} C_DIS
   LIN {X -1.974, Y 27.154, Z 20.400} C_DIS
   LIN {X -1.907, Y 26.566, Z 20.400} C_DIS
   LIN {X -1.710, Y 23.467, Z 20.400} C_DIS
   LIN {X -1.513, Y 20.654, Z 20.400} C_DIS
   LIN {X -1.522, Y 19.670, Z 20.400} C_DIS
   LIN {X -1.599, Y 14.795, Z 20.400} C_DIS
   LIN {X -1.807, Y 11.939, Z 20.400} C_DIS
   LIN {X -1.889, Y 11.154, Z 20.400} C_DIS
   LIN {X -2.251, Y 8.230, Z 20.400} C_DIS
   LIN {X -2.428, Y 7.182, Z 20.400} C_DIS
   LIN {X -3.203, Y 3.088, Z 20.400} C_DIS
   LIN {X -3.743, Y 0.797, Z 20.400} C_DIS
   LIN {X -4.850, Y -2.867, Z 20.400} C_DIS
   LIN {X -5.808, Y -5.941, Z 20.400} C_DIS
   LIN {X -6.890, Y -8.650, Z 20.400} C_DIS
   LIN {X -7.580, Y -10.388, Z 20.400} C_DIS
   LIN {X -7.911, Y -11.094, Z 20.400} C_DIS
   LIN {X -9.122, Y -13.599, Z 20.400} C_DIS
   LIN {X -9.747, Y -14.910, Z 20.400} C_DIS
   LIN {X -10.180, Y -15.697, Z 20.400} C_DIS
   LIN {X -11.623, Y -18.287, Z 20.400} C_DIS
   LIN {X -12.704, Y -21.170, Z 20.400} C_DIS
   LIN {X -12.733, Y -21.417, Z 20.400} C_DIS
   LIN {X -12.643, Y -24.966, Z 20.400} C_DIS
   LIN {X -11.864, Y -26.805, Z 20.400} C_DIS
   LIN {X -11.493, Y -27.693, Z 20.400} C_DIS
   LIN {X -10.625, Y -28.674, Z 20.400} C_DIS
   LIN {X -9.425, Y -29.953, Z 20.400} C_DIS
   LIN {X -8.708, Y -30.346, Z 20.400} C_DIS
   LIN {X -7.323, Y -31.177, Z 20.400} C_DIS
   LIN {X -5.444, Y -31.708, Z 20.400} C_DIS
   LIN {X -5.280, Y -31.722, Z 20.400} C_DIS
   LIN {X -2.413, Y -31.715, Z 20.400} C_DIS
   LIN {X 0.509, Y -30.506, Z 20.400} C_DIS
   LIN {X 1.267, Y -30.204, Z 20.400} C_DIS
   LIN {X 2.057, Y -29.414, Z 20.400} C_DIS
   LIN {X 3.476, Y -28.005, Z 20.400} C_DIS
   LIN {X 4.034, Y -26.878, Z 20.400} C_DIS
   LIN {X 4.788, Y -25.298, Z 20.400}
   LaserEnd_Ext()
   LIN {X -1.755, Y -30.360, Z 20.400}
   LaserStart_Ext()
   LIN {X -6.536, Y -30.360, Z 20.400}
   LaserEnd_Ext()
   LIN {X -8.426, Y -29.360, Z 20.400}
   LaserStart_Ext()
   LIN {X 0.683, Y -29.360, Z 20.400}
   LaserEnd_Ext()
   LIN {X 1.699, Y -28.360, Z 20.400}
   LaserStart_Ext()
   LIN {X -1.560, Y -28.360, Z 20.400}
   LaserEnd_Ext()
   LIN {X -6.178, Y -28.360, Z 20.400}
   LaserStart_Ext()
   LIN {X -9.548, Y -28.360, Z 20.400}
   LaserEnd_Ext()
   LIN {X -10.453, Y -27.360, Z 20.400}
   LaserStart_Ext()
   LIN {X -7.686, Y -27.360, Z 20.400}
   LaserEnd_Ext()
   LIN {X -0.191, Y -27.360, Z 20.400}
   LaserStart_Ext()
   LIN {X 2.679, Y -27.360, Z 20.400}
   LaserEnd_Ext()
   LIN {X 3.174, Y -26.360, Z 20.400}
   LaserStart_Ext()
   LIN {X 0.819, Y -26.360, Z 20.400}
   LaserEnd_Ext()
   LIN {X -8.676, Y -26.360, Z 20.400}
   LaserStart_Ext()
   LIN {X -10.967, Y -26.360, Z 20.400}
   LaserEnd_Ext()
   LIN {X -11.390, Y -25.360, Z 20.400}
   LaserStart_Ext()
   LIN {X -9.243, Y -25.360, Z 20.400}
   LaserEnd_Ext()
   LIN {X 1.459, Y -25.360, Z 20.400}
   LaserStart_Ext()
   LIN {X 3.651, Y -25.360, Z 20.400}
   LaserEnd_Ext()
   LIN {X 4.008, Y -24.360, Z 20.400}
   LaserStart_Ext()
   LIN {X 1.925, Y -24.360, Z 20.400}
   LaserEnd_Ext()
   LIN {X -9.666, Y -24.360, Z 20.400}
   LaserStart_Ext()
   LIN {X -11.658, Y -24.360, Z 20.400}
   LaserEnd_Ext()
   LIN {X -11.683, Y -23.360, Z 20.400}
   LaserStart_Ext()
   LIN {X -9.811, Y -23.360, Z 20.400}
   LaserEnd_Ext()
   LIN {X 1.983, Y -23.360, Z 20.400}
   LaserStart_Ext()
   LIN {X 4.282, Y -23.360, Z 20.400}
   LaserEnd_Ext()
   LIN {X 4.555, Y -22.360, Z 20.400}
   LaserStart_Ext()
   LIN {X 2.023, Y -22.360, Z 20.400}
   LaserEnd_Ext()
   LIN {X -9.804, Y -22.360, Z 20.400}
   LaserStart_Ext()
   LIN {X -11.709, Y -22.360, Z 20.400}
   LaserEnd_Ext()
   LIN {X -11.708, Y -21.360, Z 20.400}
   LaserStart_Ext()
   LIN {X -9.561, Y -21.360, Z 20.400}
   LaserEnd_Ext()
   LIN {X 1.926, Y -21.360, Z 20.400}
   LaserStart_Ext()
   LIN {X 4.811, Y -21.360, Z 20.400}
   LaserEnd_Ext()
   LIN {X 5.055, Y -20.360, Z 20.400}
   LaserStart_Ext()
   LIN {X 1.433, Y -20.360, Z 20.400}
   LaserEnd_Ext()
   LIN {X -9.315, Y -20.360, Z 20.400}
   LaserStart_Ext()
   LIN {X -11.333, Y -20.360, Z 20.400}
   LaserEnd_Ext()
   LIN {X -10.958, Y -19.360, Z 20.400}
   LaserStart_Ext()
   LIN {X -8.692, Y -19.360, Z 20.400}
   LaserEnd_Ext()
   LIN {X 0.954, Y -19.360, Z 20.400}
   LaserStart_Ext()
   LIN {X 5.299, Y -19.360, Z 20.400}
   LaserEnd_Ext()
   LIN {X 5.527, Y -18.360, Z 20.400}
   LaserStart_Ext()
   LIN {X -0.001, Y -18.360, Z 20.400}
   LaserEnd_Ext()
   LIN {X -7.730, Y -18.360, Z 20.400}
   LaserStart_Ext()
   LIN {X -10.519, Y -18.360, Z 20.400}
   LaserEnd_Ext()
   LIN {X -9.962, Y -17.360, Z 20.400}
   LaserStart_Ext()
   LIN {X -6.307, Y -17.360, Z 20.400}
   LaserEnd_Ext()
   LIN {X -1.375, Y -17.360, Z 20.400}
   LaserStart_Ext()
   LIN {X 5.737, Y -17.360, Z 20.400}
   LaserEnd_Ext()
   LIN {X 5.947, Y -16.360, Z 20.400}
   LaserStart_Ext()
   LIN {X -9.404, Y -16.360, Z 20.400}
   LaserEnd_Ext()
   LIN {X -8.855, Y -15.360, Z 20.400}
   LaserStart_Ext()
   LIN {X 6.156, Y -15.360, Z 20.400}
   LaserEnd_Ext()
   LIN {X 6.334, Y -14.360, Z 20.400}
   LaserStart_Ext()
   LIN {X -8.377, Y -14.360, Z 20.400}
   LaserEnd_Ext()
   LIN {X -7.896, Y -13.360, Z 20.400}
   LaserStart_Ext()
   LIN {X 6.501, Y -13.360, Z 20.400}
   LaserEnd_Ext()
   LIN {X 6.670, Y -12.360, Z 20.400}
   LaserStart_Ext()
   LIN {X -7.413, Y -12.360, Z 20.400}
   LaserEnd_Ext()
   LIN {X -6.931, Y -11.360, Z 20.400}
   LaserStart_Ext()
   LIN {X 6.838, Y -11.360, Z 20.400}
   LaserEnd_Ext()
   LIN {X 7.007, Y -10.360, Z 20.400}
   LaserStart_Ext()
   LIN {X -6.493, Y -10.360, Z 20.400}
   LaserEnd_Ext()
   LIN {X -6.096, Y -9.360, Z 20.400}
   LaserStart_Ext()
   LIN {X 7.142, Y -9.360, Z 20.400}
   LaserEnd_Ext()
   LIN {X 7.256, Y -8.360, Z 20.400}
   LaserStart_Ext()
   LIN {X -5.697, Y -8.360, Z 20.400}
   LaserEnd_Ext()
   LIN {X -5.298, Y -7.360, Z 20.400}
   LaserStart_Ext()
   LIN {X 7.369, Y -7.360, Z 20.400}
   LaserEnd_Ext()
   LIN {X 7.482, Y -6.360, Z 20.400}
   LaserStart_Ext()
   LIN {X -4.898, Y -6.360, Z 20.400}
   LaserEnd_Ext()
   LIN {X -4.579, Y -5.360, Z 20.400}
   LaserStart_Ext()
   LIN {X 7.596, Y -5.360, Z 20.400}
   LaserEnd_Ext()
   LIN {X 7.709, Y -4.360, Z 20.400}
   LaserStart_Ext()
   LIN {X -4.268, Y -4.360, Z 20.400}
   LaserEnd_Ext()
   LIN {X -3.956, Y -3.360, Z 20.400}
   LaserStart_Ext()
   LIN {X 7.801, Y -3.360, Z 20.400}
   LaserEnd_Ext()
   LIN {X 7.872, Y -2.360, Z 20.400}
   LaserStart_Ext()
   LIN {X -3.652, Y -2.360, Z 20.400}
   LaserEnd_Ext()
   LIN {X -3.350, Y -1.360, Z 20.400}
   LaserStart_Ext()
   LIN {X 7.899, Y -1.360, Z 20.400}
   LaserEnd_Ext()
   LIN {X 7.926, Y -0.360, Z 20.400}
   LaserStart_Ext()
   LIN {X -3.048, Y -0.360, Z 20.400}
   LaserEnd_Ext()
   LIN {X -2.753, Y 0.640, Z 20.400}
   LaserStart_Ext()
   LIN {X 7.953, Y 0.640, Z 20.400}
   LaserEnd_Ext()
   LIN {X 7.980, Y 1.640, Z 20.400}
   LaserStart_Ext()
   LIN {X -2.517, Y 1.640, Z 20.400}
   LaserEnd_Ext()
   LIN {X -2.281, Y 2.640, Z 20.400}
   LaserStart_Ext()
   LIN {X 8.008, Y 2.640, Z 20.400}
   LaserEnd_Ext()
   LIN {X 8.035, Y 3.640, Z 20.400}
   LaserStart_Ext()
   LIN {X -2.081, Y 3.640, Z 20.400}
   LaserEnd_Ext()
   LIN {X -1.892, Y 4.640, Z 20.400}
   LaserStart_Ext()
   LIN {X 8.062, Y 4.640, Z 20.400}
   LaserEnd_Ext()
   LIN {X 8.096, Y 5.640, Z 20.400}
   LaserStart_Ext()
   LIN {X -1.702, Y 5.640, Z 20.400}
   LaserEnd_Ext()
   LIN {X -1.513, Y 6.640, Z 20.400}
   LaserStart_Ext()
   LIN {X 8.130, Y 6.640, Z 20.400}
   LaserEnd_Ext()
   LIN {X 8.138, Y 7.640, Z 20.400}
   LaserStart_Ext()
   LIN {X -1.337, Y 7.640, Z 20.400}
   LaserEnd_Ext()
   LIN {X -1.193, Y 8.640, Z 20.400}
   LaserStart_Ext()
   LIN {X 8.100, Y 8.640, Z 20.400}
   LaserEnd_Ext()
   LIN {X 8.060, Y 9.640, Z 20.400}
   LaserStart_Ext()
   LIN {X -1.069, Y 9.640, Z 20.400}
   LaserEnd_Ext()
   LIN {X -0.945, Y 10.640, Z 20.400}
   LaserStart_Ext()
   LIN {X 8.019, Y 10.640, Z 20.400}
   LaserEnd_Ext()
   LIN {X 7.979, Y 11.640, Z 20.400}
   LaserStart_Ext()
   LIN {X -0.832, Y 11.640, Z 20.400}
   LaserEnd_Ext()
   LIN {X -0.753, Y 12.640, Z 20.400}
   LaserStart_Ext()
   LIN {X 7.930, Y 12.640, Z 20.400}
   LaserEnd_Ext()
   LIN {X 7.848, Y 13.640, Z 20.400}
   LaserStart_Ext()
   LIN {X -0.680, Y 13.640, Z 20.400}
   LaserEnd_Ext()
   LIN {X -0.608, Y 14.640, Z 20.400}
   LaserStart_Ext()
   LIN {X 7.767, Y 14.640, Z 20.400}
   LaserEnd_Ext()
   LIN {X 7.686, Y 15.640, Z 20.400}
   LaserStart_Ext()
   LIN {X -0.585, Y 15.640, Z 20.400}
   LaserEnd_Ext()
   LIN {X -0.570, Y 16.640, Z 20.400}
   LaserStart_Ext()
   LIN {X 7.584, Y 16.640, Z 20.400}
   LaserEnd_Ext()
   LIN {X 7.467, Y 17.640, Z 20.400}
   LaserStart_Ext()
   LIN {X -0.554, Y 17.640, Z 20.400}
   LaserEnd_Ext()
   LIN {X -0.538, Y 18.640, Z 20.400}
   LaserStart_Ext()
   LIN {X 7.349, Y 18.640, Z 20.400}
   LaserEnd_Ext()
   LIN {X 7.231, Y 19.640, Z 20.400}
   LaserStart_Ext()
   LIN {X -0.522, Y 19.640, Z 20.400}
   LaserEnd_Ext()
   LIN {X -0.513, Y 20.640, Z 20.400}
   LaserStart_Ext()
   LIN {X 7.100, Y 20.640, Z 20.400}
   LaserEnd_Ext()
   LIN {X 6.940, Y 21.640, Z 20.400}
   LaserStart_Ext()
   LIN {X -0.579, Y 21.640, Z 20.400}
   LaserEnd_Ext()
   LIN {X -0.649, Y 22.640, Z 20.400}
   LaserStart_Ext()
   LIN {X 6.780, Y 22.640, Z 20.400}
   LaserEnd_Ext()
   LIN {X 6.620, Y 23.640, Z 20.400}
   LaserStart_Ext()
   LIN {X -0.719, Y 23.640, Z 20.400}
   LaserEnd_Ext()
   LIN {X -0.782, Y 24.640, Z 20.400}
   LaserStart_Ext()
   LIN {X 6.449, Y 24.640, Z 20.400}
   LaserEnd_Ext()
   LIN {X 6.278, Y 25.640, Z 20.400}
   LaserStart_Ext()
   LIN {X -0.846, Y 25.640, Z 20.400}
   LaserEnd_Ext()
   LIN {X -0.910, Y 26.640, Z 20.400}
   LaserStart_Ext()
   LIN {X 6.093, Y 26.640, Z 20.400}
   LaserEnd_Ext()
   LIN {X 5.880, Y 27.640, Z 20.400}
   LaserStart_Ext()
   LIN {X -1.030, Y 27.640, Z 20.400}
   LaserEnd_Ext()
   LIN {X -1.166, Y 28.640, Z 20.400}
   LaserStart_Ext()
   LIN {X 5.668, Y 28.640, Z 20.400}
   LaserEnd_Ext()
   LIN {X 5.458, Y 29.640, Z 20.400}
   LaserStart_Ext()
   LIN {X -1.301, Y 29.640, Z 20.400}
   LaserEnd_Ext()
   LIN {X -1.449, Y 30.640, Z 20.400}
   LaserStart_Ext()
   LIN {X 5.228, Y 30.640, Z 20.400}
   LaserEnd_Ext()
   LIN {X 4.981, Y 31.640, Z 20.400}
   LaserStart_Ext()
   LIN {X -1.624, Y 31.640, Z 20.400}
   LaserEnd_Ext()
   LIN {X -1.798, Y 32.640, Z 20.400}
   LaserStart_Ext()
   LIN {X 4.733, Y 32.640, Z 20.400}
   LaserEnd_Ext()
   LIN {X 4.481, Y 33.640, Z 20.400}
   LaserStart_Ext()
   LIN {X -2.004, Y 33.640, Z 20.400}
   LaserEnd_Ext()
   LIN {X -2.213, Y 34.640, Z 20.400}
   LaserStart_Ext()
   LIN {X 4.203, Y 34.640, Z 20.400}
   LaserEnd_Ext()
   LIN {X 3.926, Y 35.640, Z 20.400}
   LaserStart_Ext()
   LIN {X -2.437, Y 35.640, Z 20.400}
   LaserEnd_Ext()
   LIN {X -2.675, Y 36.640, Z 20.400}
   LaserStart_Ext()
   LIN {X 3.637, Y 36.640, Z 20.400}
   LaserEnd_Ext()
   LIN {X 3.336, Y 37.640, Z 20.400}
   LaserStart_Ext()
   LIN {X -2.926, Y 37.640, Z 20.400}
   LaserEnd_Ext()
   LIN {X -3.044, Y 38.640, Z 20.400}
   LaserStart_Ext()
   LIN {X 3.025, Y 38.640, Z 20.400}
   LaserEnd_Ext()
   LIN {X 2.663, Y 39.640, Z 20.400}
   LaserStart_Ext()
   LIN {X -2.857, Y 39.640, Z 20.400}
   LaserEnd_Ext()
   LIN {X -2.241, Y 40.640, Z 20.400}
   LaserStart_Ext()
   LIN {X 2.007, Y 40.640, Z 20.400}
   LaserEnd_Ext()
   LIN {X 1.041, Y -24.037, Z 21.250}
   LaserStart_Ext()
   LIN {X 0.288, Y -25.541, Z 21.250} C_DIS
   LIN {X 0.123, Y -25.871, Z 21.250} C_DIS
   LIN {X -0.147, Y -26.079, Z 21.250} C_DIS
   LIN {X -1.800, Y -27.364, Z 21.250} C_DIS
   LIN {X -3.896, Y -27.784, Z 21.250} C_DIS
   LIN {X -5.929, Y -27.331, Z 21.250} C_DIS
   LIN {X -7.181, Y -26.389, Z 21.250} C_DIS
   LIN {X -7.578, Y -26.088, Z 21.250} C_DIS
   LIN {X -7.916, Y -25.491, Z 21.250} C_DIS
   LIN {X -8.569, Y -24.339, Z 21.250} C_DIS
   LIN {X -8.734, Y -23.221, Z 21.250} C_DIS
   LIN {X -8.795, Y -22.669, Z 21.250} C_DIS
   LIN {X -8.381, Y -20.941, Z 21.250} C_DIS
   LIN {X -7.962, Y -20.122, Z 21.250} C_DIS
   LIN {X -7.461, Y -19.404, Z 21.250} C_DIS
   LIN {X -6.003, Y -18.364, Z 21.250} C_DIS
   LIN {X -5.775, Y -18.201, Z 21.250} C_DIS
   LIN {X -5.394, Y -18.125, Z 21.250} C_DIS
   LIN {X -3.713, Y -17.786, Z 21.250} C_DIS
   LIN {X -1.674, Y -18.239, Z 21.250} C_DIS
   LIN {X -0.980, Y -18.765, Z 21.250} C_DIS
   LIN {X 0.017, Y -19.525, Z 21.250} C_DIS
   LIN {X 0.619, Y -20.779, Z 21.250} C_DIS
   LIN {X 1.121, Y -21.817, Z 21.250} C_DIS
   LIN {X 1.096, Y -22.691, Z 21.250} C_DIS
   LIN {X 1.041, Y -24.037, Z 21.250}
   LaserEnd_Ext()
   LIN {X 1.306, Y -30.181, Z 21.250}
   LaserStart_Ext()
   LIN {X 3.529, Y -27.957, Z 21.250} C_DIS
   LIN {X 3.643, Y -27.796, Z 21.250} C_DIS
   LIN {X 4.867, Y -25.231, Z 21.250} C_DIS
   LIN {X 5.377, Y -23.365, Z 21.250} C_DIS
   LIN {X 5.721, Y -22.081, Z 21.250} C_DIS
   LIN {X 6.084, Y -20.561, Z 21.250} C_DIS
   LIN {X 6.453, Y -19.047, Z 21.250} C_DIS
   LIN {X 6.825, Y -17.275, Z 21.250} C_DIS
   LIN {X 7.247, Y -15.227, Z 21.250} C_DIS
   LIN {X 7.952, Y -11.000, Z 21.250} C_DIS
   LIN {X 8.083, Y -10.170, Z 21.250} C_DIS
   LIN {X 8.556, Y -5.899, Z 21.250} C_DIS
   LIN {X 8.806, Y -3.689, Z 21.250} C_DIS
   LIN {X 8.833, Y -3.368, Z 21.250} C_DIS
   LIN {X 8.875, Y -1.822, Z 21.250} C_DIS
   LIN {X 9.157, Y 6.302, Z 21.250} C_DIS
   LIN {X 9.095, Y 8.689, Z 21.250} C_DIS
   LIN {X 8.939, Y 12.531, Z 21.250} C_DIS
   LIN {X 8.690, Y 15.600, Z 21.250} C_DIS
   LIN {X 8.232, Y 19.525, Z 21.250} C_DIS
   LIN {X 8.097, Y 20.670, Z 21.250} C_DIS
   LIN {X 7.858, Y 22.163, Z 21.250} C_DIS
   LIN {X 7.107, Y 26.558, Z 21.250} C_DIS
   LIN {X 6.369, Y 30.026, Z 21.250} C_DIS
   LIN {X 6.330, Y 30.199, Z 21.250} C_DIS
   LIN {X 6.288, Y 30.364, Z 21.250} C_DIS
   LIN {X 6.132, Y 30.992, Z 21.250} C_DIS
   LIN {X 5.435, Y 33.799, Z 21.250} C_DIS
   LIN {X 5.154, Y 34.810, Z 21.250} C_DIS
   LIN {X 4.723, Y 36.350, Z 21.250} C_DIS
   LIN {X 4.142, Y 38.269, Z 21.250} C_DIS
   LIN {X 4.094, Y 38.426, Z 21.250} C_DIS
   LIN {X 4.040, Y 38.594, Z 21.250} C_DIS
   LIN {X 3.617, Y 39.912, Z 21.250} C_DIS
   LIN {X 3.137, Y 40.788, Z 21.250} C_DIS
   LIN {X 2.908, Y 41.203, Z 21.250} C_DIS
   LIN {X 2.326, Y 41.661, Z 21.250} C_DIS
   LIN {X 1.540, Y 42.281, Z 21.250} C_DIS
   LIN {X 0.904, Y 42.431, Z 21.250} C_DIS
   LIN {X -0.161, Y 42.678, Z 21.250} C_DIS
   LIN {X -1.976, Y 42.059, Z 21.250} C_DIS
   LIN {X -2.671, Y 41.808, Z 21.250} C_DIS
   LIN {X -2.965, Y 41.436, Z 21.250} C_DIS
   LIN {X -3.752, Y 40.469, Z 21.250} C_DIS
   LIN {X -3.995, Y 39.639, Z 21.250} C_DIS
   LIN {X -4.140, Y 39.125, Z 21.250} C_DIS
   LIN {X -4.077, Y 38.414, Z 21.250} C_DIS
   LIN {X -4.017, Y 37.659, Z 21.250} C_DIS
   LIN {X -3.911, Y 37.244, Z 21.250} C_DIS
   LIN {X -3.709, Y 36.446, Z 21.250} C_DIS
   LIN {X -3.346, Y 34.932, Z 21.250} C_DIS
   LIN {X -3.319, Y 34.808, Z 21.250} C_DIS
   LIN {X -2.847, Y 32.569, Z 21.250} C_DIS
   LIN {X -2.531, Y 30.790, Z 21.250} C_DIS
   LIN {X -2.433, Y 30.233, Z 21.250} C_DIS
   LIN {X -2.114, Y 27.869, Z 21.250} C_DIS
   LIN {X -1.957, Y 26.721, Z 21.250} C_DIS
   LIN {X -1.922, Y 26.262, Z 21.250} C_DIS
   LIN {X -1.545, Y 20.876, Z 21.250} C_DIS
   LIN {X -1.565, Y 18.659, Z 21.250} C_DIS
   LIN {X -1.632, Y 14.486, Z 21.250} C_DIS
   LIN {X -1.809, Y 12.041, Z 21.250} C_DIS
   LIN {X -1.960, Y 10.607, Z 21.250} C_DIS
   LIN {X -2.240, Y 8.345, Z 21.250} C_DIS
   LIN {X -2.600, Y 6.212, Z 21.250} C_DIS
   LIN {X -3.143, Y 3.344, Z 21.250} C_DIS
   LIN {X -3.844, Y 0.372, Z 21.250} C_DIS
   LIN {X -4.413, Y -1.514, Z 21.250} C_DIS
   LIN {X -5.827, Y -6.049, Z 21.250} C_DIS
   LIN {X -7.423, Y -10.045, Z 21.250} C_DIS
   LIN {X -7.614, Y -10.527, Z 21.250} C_DIS
   LIN {X -7.706, Y -10.722, Z 21.250} C_DIS
   LIN {X -8.041, Y -11.417, Z 21.250} C_DIS
   LIN {X -9.684, Y -14.861, Z 21.250} C_DIS
   LIN {X -10.821, Y -16.931, Z 21.250} C_DIS
   LIN {X -11.561, Y -18.258, Z 21.250} C_DIS
   LIN {X -12.154, Y -19.841, Z 21.250} C_DIS
   LIN {X -12.667, Y -21.229, Z 21.250} C_DIS
   LIN {X -12.634, Y -22.253, Z 21.250} C_DIS
   LIN {X -12.565, Y -24.939, Z 21.250} C_DIS
   LIN {X -11.485, Y -27.490, Z 21.250} C_DIS
   LIN {X -11.412, Y -27.662, Z 21.250} C_DIS
   LIN {X -11.237, Y -27.837, Z 21.250} C_DIS
   LIN {X -9.172, Y -30.038, Z 21.250} C_DIS
   LIN {X -7.734, Y -30.826, Z 21.250} C_DIS
   LIN {X -7.170, Y -31.164, Z 21.250} C_DIS
   LIN {X -6.353, Y -31.395, Z 21.250} C_DIS
   LIN {X -5.377, Y -31.666, Z 21.250} C_DIS
   LIN {X -3.910, Y -31.683, Z 21.250} C_DIS
   LIN {X -2.403, Y -31.679, Z 21.250} C_DIS
   LIN {X -0.978, Y -31.089, Z 21.250} C_DIS
   LIN {X 1.306, Y -30.181, Z 21.250}
   LaserEnd_Ext()
   LIN {X 7.602, Y -5.434, Z 21.250}
   LaserStart_Ext()
   LIN {X 7.602, Y 16.295, Z 21.250}
   LaserEnd_Ext()
   LIN {X 6.602, Y 23.578, Z 21.250}
   LaserStart_Ext()
   LIN {X 6.602, Y -13.014, Z 21.250}
   LaserEnd_Ext()
   LIN {X 5.602, Y -18.234, Z 21.250}
   LaserStart_Ext()
   LIN {X 5.602, Y 28.826, Z 21.250}
   LaserEnd_Ext()
   LIN {X 4.602, Y 33.005, Z 21.250}
   LaserStart_Ext()
   LIN {X 4.602, Y -22.394, Z 21.250}
   LaserEnd_Ext()
   LIN {X 3.602, Y -25.560, Z 21.250}
   LaserStart_Ext()
   LIN {X 3.602, Y 36.602, Z 21.250}
   LaserEnd_Ext()
   LIN {X 2.602, Y 39.683, Z 21.250}
   LaserStart_Ext()
   LIN {X 2.602, Y -27.470, Z 21.250}
   LaserEnd_Ext()
   LIN {X 1.602, Y -28.471, Z 21.250}
   LaserStart_Ext()
   LIN {X 1.602, Y -25.151, Z 21.250}
   LaserEnd_Ext()
   LIN {X 1.602, Y -20.515, Z 21.250}
   LaserStart_Ext()
   LIN {X 1.602, Y 40.958, Z 21.250}
   LaserEnd_Ext()
   LIN {X 0.602, Y 41.474, Z 21.250}
   LaserStart_Ext()
   LIN {X 0.602, Y -18.714, Z 21.250}
   LaserEnd_Ext()
   LIN {X 0.602, Y -26.765, Z 21.250}
   LaserStart_Ext()
   LIN {X 0.602, Y -29.385, Z 21.250}
   LaserEnd_Ext()
   LIN {X -0.398, Y -29.783, Z 21.250}
   LaserStart_Ext()
   LIN {X -0.398, Y -27.541, Z 21.250}
   LaserEnd_Ext()
   LIN {X -0.398, Y -17.951, Z 21.250}
   LaserStart_Ext()
   LIN {X -0.398, Y 41.541, Z 21.250}
   LaserEnd_Ext()
   LIN {X -1.398, Y 41.199, Z 21.250}
   LaserStart_Ext()
   LIN {X -1.398, Y 30.039, Z 21.250}
   LaserEnd_Ext()
   LIN {X -1.398, Y 7.327, Z 21.250}
   LaserStart_Ext()
   LIN {X -1.398, Y -17.280, Z 21.250}
   LaserEnd_Ext()
   LIN {X -1.398, Y -28.279, Z 21.250}
   LaserStart_Ext()
   LIN {X -1.398, Y -30.181, Z 21.250}
   LaserEnd_Ext()
   LIN {X -2.398, Y -30.595, Z 21.250}
   LaserStart_Ext()
   LIN {X -2.398, Y -28.504, Z 21.250}
   LaserEnd_Ext()
   LIN {X -2.398, Y -17.054, Z 21.250}
   LaserStart_Ext()
   LIN {X -2.398, Y 2.146, Z 21.250}
   LaserEnd_Ext()
   LIN {X -2.398, Y 35.265, Z 21.250}
   LaserStart_Ext()
   LIN {X -2.398, Y 40.548, Z 21.250}
   LaserEnd_Ext()
   LIN {X -3.398, Y -1.611, Z 21.250}
   LaserStart_Ext()
   LIN {X -3.398, Y -16.832, Z 21.250}
   LaserEnd_Ext()
   LIN {X -3.398, Y -28.704, Z 21.250}
   LaserStart_Ext()
   LIN {X -3.398, Y -30.681, Z 21.250}
   LaserEnd_Ext()
   LIN {X -4.398, Y -30.677, Z 21.250}
   LaserStart_Ext()
   LIN {X -4.398, Y -28.703, Z 21.250}
   LaserEnd_Ext()
   LIN {X -4.398, Y -16.904, Z 21.250}
   LaserStart_Ext()
   LIN {X -4.398, Y -4.826, Z 21.250}
   LaserEnd_Ext()
   LIN {X -5.398, Y -7.672, Z 21.250}
   LaserStart_Ext()
   LIN {X -5.398, Y -17.106, Z 21.250}
   LaserEnd_Ext()
   LIN {X -5.398, Y -28.476, Z 21.250}
   LaserStart_Ext()
   LIN {X -5.398, Y -30.622, Z 21.250}
   LaserEnd_Ext()
   LIN {X -6.398, Y -30.343, Z 21.250}
   LaserStart_Ext()
   LIN {X -6.398, Y -28.212, Z 21.250}
   LaserEnd_Ext()
   LIN {X -6.398, Y -17.417, Z 21.250}
   LaserStart_Ext()
   LIN {X -6.398, Y -10.176, Z 21.250}
   LaserEnd_Ext()
   LIN {X -7.398, Y -12.391, Z 21.250}
   LaserStart_Ext()
   LIN {X -7.398, Y -18.131, Z 21.250}
   LaserEnd_Ext()
   LIN {X -7.398, Y -27.477, Z 21.250}
   LaserStart_Ext()
   LIN {X -7.398, Y -29.869, Z 21.250}
   LaserEnd_Ext()
   LIN {X -8.398, Y -29.322, Z 21.250}
   LaserStart_Ext()
   LIN {X -8.398, Y -26.660, Z 21.250}
   LaserEnd_Ext()
   LIN {X -8.398, Y -19.000, Z 21.250}
   LaserStart_Ext()
   LIN {X -8.398, Y -14.488, Z 21.250}
   LaserEnd_Ext()
   LIN {X -9.398, Y -16.418, Z 21.250}
   LaserStart_Ext()
   LIN {X -9.398, Y -20.892, Z 21.250}
   LaserEnd_Ext()
   LIN {X -9.398, Y -24.905, Z 21.250}
   LaserStart_Ext()
   LIN {X -9.398, Y -28.336, Z 21.250}
   LaserEnd_Ext()
   LIN {X -10.398, Y -27.270, Z 21.250}
   LaserStart_Ext()
   LIN {X -10.398, Y -18.226, Z 21.250}
   LaserEnd_Ext()
   LIN {X -11.398, Y -20.680, Z 21.250}
   LaserStart_Ext()
   LIN {X -11.398, Y -25.131, Z 21.250}
   LaserEnd_Ext()
   LIN {X 0.158, Y -25.874, Z 22.100}
   LaserStart_Ext()
   LIN {X -1.519, Y -27.166, Z 22.100} C_DIS
   LIN {X -1.703, Y -27.308, Z 22.100} C_DIS
   LIN {X -1.940, Y -27.356, Z 22.100} C_DIS
   LIN {X -3.829, Y -27.741, Z 22.100} C_DIS
   LIN {X -5.097, Y -27.459, Z 22.100} C_DIS
   LIN {X -5.844, Y -27.290, Z 22.100} C_DIS
   LIN {X -6.628, Y -26.700, Z 22.100} C_DIS
   LIN {X -7.496, Y -26.050, Z 22.100} C_DIS
   LIN {X -7.900, Y -25.340, Z 22.100} C_DIS
   LIN {X -8.496, Y -24.289, Z 22.100} C_DIS
   LIN {X -8.577, Y -23.742, Z 22.100} C_DIS
   LIN {X -8.713, Y -22.503, Z 22.100} C_DIS
   LIN {X -8.424, Y -21.293, Z 22.100} C_DIS
   LIN {X -7.557, Y -19.602, Z 22.100} C_DIS
   LIN {X -7.387, Y -19.359, Z 22.100} C_DIS
   LIN {X -6.892, Y -19.006, Z 22.100} C_DIS
   LIN {X -5.692, Y -18.151, Z 22.100} C_DIS
   LIN {X -3.685, Y -17.751, Z 22.100} C_DIS
   LIN {X -1.610, Y -18.188, Z 22.100} C_DIS
   LIN {X -0.181, Y -19.271, Z 22.100} C_DIS
   LIN {X 0.084, Y -19.470, Z 22.100} C_DIS
   LIN {X 0.271, Y -19.853, Z 22.100} C_DIS
   LIN {X 1.193, Y -21.759, Z 22.100} C_DIS
   LIN {X 1.134, Y -23.821, Z 22.100} C_DIS
   LIN {X 1.131, Y -23.934, Z 22.100} C_DIS
   LIN {X 1.085, Y -24.025, Z 22.100} C_DIS
   LIN {X 0.158, Y -25.874, Z 22.100}
   LaserEnd_Ext()
   LIN {X -1.703, Y 22.894, Z 22.100}
   LaserStart_Ext()
   LIN {X -1.578, Y 21.098, Z 22.100} C_DIS
   LIN {X -1.609, Y 17.648, Z 22.100} C_DIS
   LIN {X -1.664, Y 14.177, Z 22.100} C_DIS
   LIN {X -1.812, Y 12.143, Z 22.100} C_DIS
   LIN {X -2.031, Y 10.060, Z 22.100} C_DIS
   LIN {X -2.230, Y 8.460, Z 22.100} C_DIS
   LIN {X -2.773, Y 5.242, Z 22.100} C_DIS
   LIN {X -3.083, Y 3.600, Z 22.100} C_DIS
   LIN {X -3.944, Y -0.054, Z 22.100} C_DIS
   LIN {X -3.977, Y -0.162, Z 22.100} C_DIS
   LIN {X -5.846, Y -6.157, Z 22.100} C_DIS
   LIN {X -7.266, Y -9.714, Z 22.100} C_DIS
   LIN {X -7.612, Y -10.588, Z 22.100} C_DIS
   LIN {X -8.014, Y -11.444, Z 22.100} C_DIS
   LIN {X -9.620, Y -14.813, Z 22.100} C_DIS
   LIN {X -11.462, Y -18.165, Z 22.100} C_DIS
   LIN {X -11.527, Y -18.307, Z 22.100} C_DIS
   LIN {X -12.597, Y -21.203, Z 22.100} C_DIS
   LIN {X -12.527, Y -23.340, Z 22.100} C_DIS
   LIN {X -12.487, Y -24.913, Z 22.100} C_DIS
   LIN {X -11.855, Y -26.407, Z 22.100} C_DIS
   LIN {X -11.325, Y -27.634, Z 22.100} C_DIS
   LIN {X -10.075, Y -28.892, Z 22.100} C_DIS
   LIN {X -8.920, Y -30.124, Z 22.100} C_DIS
   LIN {X -7.369, Y -30.972, Z 22.100} C_DIS
   LIN {X -6.872, Y -31.190, Z 22.100} C_DIS
   LIN {X -5.362, Y -31.609, Z 22.100} C_DIS
   LIN {X -2.448, Y -31.642, Z 22.100} C_DIS
   LIN {X -2.169, Y -31.556, Z 22.100} C_DIS
   LIN {X 1.345, Y -30.158, Z 22.100} C_DIS
   LIN {X 2.309, Y -29.194, Z 22.100} C_DIS
   LIN {X 3.549, Y -28.003, Z 22.100} C_DIS
   LIN {X 4.487, Y -26.126, Z 22.100} C_DIS
   LIN {X 4.946, Y -25.164, Z 22.100} C_DIS
   LIN {X 5.137, Y -24.465, Z 22.100} C_DIS
   LIN {X 5.793, Y -22.012, Z 22.100} C_DIS
   LIN {X 6.487, Y -19.107, Z 22.100} C_DIS
   LIN {X 6.525, Y -18.939, Z 22.100} C_DIS
   LIN {X 7.298, Y -15.180, Z 22.100} C_DIS
   LIN {X 7.745, Y -12.502, Z 22.100} C_DIS
   LIN {X 8.141, Y -9.995, Z 22.100} C_DIS
   LIN {X 8.731, Y -4.664, Z 22.100} C_DIS
   LIN {X 8.840, Y -3.592, Z 22.100} C_DIS
   LIN {X 8.875, Y -2.892, Z 22.100} C_DIS
   LIN {X 9.164, Y 5.423, Z 22.100} C_DIS
   LIN {X 9.059, Y 9.477, Z 22.100} C_DIS
   LIN {X 8.934, Y 12.572, Z 22.100} C_DIS
   LIN {X 8.733, Y 15.044, Z 22.100} C_DIS
   LIN {X 8.091, Y 20.542, Z 22.100} C_DIS
   LIN {X 8.045, Y 20.918, Z 22.100} C_DIS
   LIN {X 7.988, Y 21.237, Z 22.100} C_DIS
   LIN {X 7.070, Y 26.611, Z 22.100} C_DIS
   LIN {X 6.548, Y 29.063, Z 22.100} C_DIS
   LIN {X 6.254, Y 30.377, Z 22.100} C_DIS
   LIN {X 5.934, Y 31.634, Z 22.100} C_DIS
   LIN {X 5.398, Y 33.789, Z 22.100} C_DIS
   LIN {X 4.969, Y 35.315, Z 22.100} C_DIS
   LIN {X 4.690, Y 36.310, Z 22.100} C_DIS
   LIN {X 4.551, Y 36.768, Z 22.100} C_DIS
   LIN {X 4.013, Y 38.527, Z 22.100} C_DIS
   LIN {X 3.640, Y 39.683, Z 22.100} C_DIS
   LIN {X 3.544, Y 39.975, Z 22.100} C_DIS
   LIN {X 3.358, Y 40.312, Z 22.100} C_DIS
   LIN {X 2.833, Y 41.265, Z 22.100} C_DIS
   LIN {X 2.044, Y 41.885, Z 22.100} C_DIS
   LIN {X 1.462, Y 42.339, Z 22.100} C_DIS
   LIN {X 0.071, Y 42.660, Z 22.100} C_DIS
   LIN {X -0.240, Y 42.732, Z 22.100} C_DIS
   LIN {X -0.588, Y 42.613, Z 22.100} C_DIS
   LIN {X -2.634, Y 41.944, Z 22.100} C_DIS
   LIN {X -3.335, Y 41.119, Z 22.100} C_DIS
   LIN {X -3.825, Y 40.516, Z 22.100} C_DIS
   LIN {X -4.011, Y 39.880, Z 22.100} C_DIS
   LIN {X -4.211, Y 39.164, Z 22.100} C_DIS
   LIN {X -4.141, Y 38.414, Z 22.100} C_DIS
   LIN {X -4.084, Y 37.704, Z 22.100} C_DIS
   LIN {X -3.859, Y 36.826, Z 22.100} C_DIS
   LIN {X -3.773, Y 36.492, Z 22.100} C_DIS
   LIN {X -3.709, Y 36.226, Z 22.100} C_DIS
   LIN {X -3.397, Y 34.936, Z 22.100} C_DIS
   LIN {X -2.929, Y 32.746, Z 22.100} C_DIS
   LIN {X -2.902, Y 32.617, Z 22.100} C_DIS
   LIN {X -2.872, Y 32.446, Z 22.100} C_DIS
   LIN {X -2.483, Y 30.282, Z 22.100} C_DIS
   LIN {X -2.250, Y 28.621, Z 22.100} C_DIS
   LIN {X -1.998, Y 26.771, Z 22.100} C_DIS
   LIN {X -1.703, Y 22.894, Z 22.100}
   LaserEnd_Ext()
   LIN {X -0.709, Y 41.522, Z 22.100}
   LaserStart_Ext()
   LIN {X 0.557, Y 41.522, Z 22.100}
   LaserEnd_Ext()
   LIN {X 2.100, Y 40.522, Z 22.100}
   LaserStart_Ext()
   LIN {X -2.529, Y 40.522, Z 22.100}
   LaserEnd_Ext()
   LIN {X -3.073, Y 39.522, Z 22.100}
   LaserStart_Ext()
   LIN {X 2.640, Y 39.522, Z 22.100}
   LaserEnd_Ext()
   LIN {X 2.964, Y 38.522, Z 22.100}
   LaserStart_Ext()
   LIN {X -3.147, Y 38.522, Z 22.100}
   LaserEnd_Ext()
   LIN {X -3.005, Y 37.522, Z 22.100}
   LaserStart_Ext()
   LIN {X 3.275, Y 37.522, Z 22.100}
   LaserEnd_Ext()
   LIN {X 3.581, Y 36.522, Z 22.100}
   LaserStart_Ext()
   LIN {X -2.751, Y 36.522, Z 22.100}
   LaserEnd_Ext()
   LIN {X -2.510, Y 35.522, Z 22.100}
   LaserStart_Ext()
   LIN {X 3.872, Y 35.522, Z 22.100}
   LaserEnd_Ext()
   LIN {X 4.153, Y 34.522, Z 22.100}
   LaserStart_Ext()
   LIN {X -2.286, Y 34.522, Z 22.100}
   LaserEnd_Ext()
   LIN {X -2.072, Y 33.522, Z 22.100}
   LaserStart_Ext()
   LIN {X 4.434, Y 33.522, Z 22.100}
   LaserEnd_Ext()
   LIN {X 4.683, Y 32.522, Z 22.100}
   LaserStart_Ext()
   LIN {X -1.869, Y 32.522, Z 22.100}
   LaserEnd_Ext()
   LIN {X -1.690, Y 31.522, Z 22.100}
   LaserStart_Ext()
   LIN {X 4.931, Y 31.522, Z 22.100}
   LaserEnd_Ext()
   LIN {X 5.185, Y 30.522, Z 22.100}
   LaserStart_Ext()
   LIN {X -1.510, Y 30.522, Z 22.100}
   LaserEnd_Ext()
   LIN {X -1.367, Y 29.522, Z 22.100}
   LaserStart_Ext()
   LIN {X 5.420, Y 29.522, Z 22.100}
   LaserEnd_Ext()
   LIN {X 5.641, Y 28.522, Z 22.100}
   LaserStart_Ext()
   LIN {X -1.228, Y 28.522, Z 22.100}
   LaserEnd_Ext()
   LIN {X -1.091, Y 27.522, Z 22.100}
   LaserStart_Ext()
   LIN {X 5.853, Y 27.522, Z 22.100}
   LaserEnd_Ext()
   LIN {X 6.066, Y 26.522, Z 22.100}
   LaserStart_Ext()
   LIN {X -0.977, Y 26.522, Z 22.100}
   LaserEnd_Ext()
   LIN {X -0.900, Y 25.522, Z 22.100}
   LaserStart_Ext()
   LIN {X 6.241, Y 25.522, Z 22.100}
   LaserEnd_Ext()
   LIN {X 6.412, Y 24.522, Z 22.100}
   LaserStart_Ext()
   LIN {X -0.824, Y 24.522, Z 22.100}
   LaserEnd_Ext()
   LIN {X -0.748, Y 23.522, Z 22.100}
   LaserStart_Ext()
   LIN {X 6.583, Y 23.522, Z 22.100}
   LaserEnd_Ext()
   LIN {X 6.754, Y 22.522, Z 22.100}
   LaserStart_Ext()
   LIN {X -0.675, Y 22.522, Z 22.100}
   LaserEnd_Ext()
   LIN {X -0.605, Y 21.522, Z 22.100}
   LaserStart_Ext()
   LIN {X 6.925, Y 21.522, Z 22.100}
   LaserEnd_Ext()
   LIN {X 7.086, Y 20.522, Z 22.100}
   LaserStart_Ext()
   LIN {X -0.583, Y 20.522, Z 22.100}
   LaserEnd_Ext()
   LIN {X -0.592, Y 19.522, Z 22.100}
   LaserStart_Ext()
   LIN {X 7.203, Y 19.522, Z 22.100}
   LaserEnd_Ext()
   LIN {X 7.320, Y 18.522, Z 22.100}
   LaserStart_Ext()
   LIN {X -0.601, Y 18.522, Z 22.100}
   LaserEnd_Ext()
   LIN {X -0.611, Y 17.522, Z 22.100}
   LaserStart_Ext()
   LIN {X 7.437, Y 17.522, Z 22.100}
   LaserEnd_Ext()
   LIN {X 7.553, Y 16.522, Z 22.100}
   LaserStart_Ext()
   LIN {X -0.627, Y 16.522, Z 22.100}
   LaserEnd_Ext()
   LIN {X -0.643, Y 15.522, Z 22.100}
   LaserStart_Ext()
   LIN {X 7.670, Y 15.522, Z 22.100}
   LaserEnd_Ext()
   LIN {X 7.772, Y 14.522, Z 22.100}
   LaserStart_Ext()
   LIN {X -0.659, Y 14.522, Z 22.100}
   LaserEnd_Ext()
   LIN {X -0.709, Y 13.522, Z 22.100}
   LaserStart_Ext()
   LIN {X 7.853, Y 13.522, Z 22.100}
   LaserEnd_Ext()
   LIN {X 7.935, Y 12.522, Z 22.100}
   LaserStart_Ext()
   LIN {X -0.782, Y 12.522, Z 22.100}
   LaserEnd_Ext()
   LIN {X -0.872, Y 11.522, Z 22.100}
   LaserStart_Ext()
   LIN {X 7.976, Y 11.522, Z 22.100}
   LaserEnd_Ext()
   LIN {X 8.016, Y 10.522, Z 22.100}
   LaserStart_Ext()
   LIN {X -0.977, Y 10.522, Z 22.100}
   LaserEnd_Ext()
   LIN {X -1.091, Y 9.522, Z 22.100}
   LaserStart_Ext()
   LIN {X 8.057, Y 9.522, Z 22.100}
   LaserEnd_Ext()
   LIN {X 8.084, Y 8.522, Z 22.100}
   LaserStart_Ext()
   LIN {X -1.214, Y 8.522, Z 22.100}
   LaserEnd_Ext()
   LIN {X -1.374, Y 7.522, Z 22.100}
   LaserStart_Ext()
   LIN {X 8.109, Y 7.522, Z 22.100}
   LaserEnd_Ext()
   LIN {X 8.135, Y 6.522, Z 22.100}
   LaserStart_Ext()
   LIN {X -1.543, Y 6.522, Z 22.100}
   LaserEnd_Ext()
   LIN {X -1.711, Y 5.522, Z 22.100}
   LaserStart_Ext()
   LIN {X 8.161, Y 5.522, Z 22.100}
   LaserEnd_Ext()
   LIN {X 8.132, Y 4.522, Z 22.100}
   LaserStart_Ext()
   LIN {X -1.891, Y 4.522, Z 22.100}
   LaserEnd_Ext()
   LIN {X -2.080, Y 3.522, Z 22.100}
   LaserStart_Ext()
   LIN {X 8.097, Y 3.522, Z 22.100}
   LaserEnd_Ext()
   LIN {X 8.062, Y 2.522, Z 22.100}
   LaserStart_Ext()
   LIN {X -2.310, Y 2.522, Z 22.100}
   LaserEnd_Ext()
   LIN {X -2.546, Y 1.522, Z 22.100}
   LaserStart_Ext()
   LIN {X 8.028, Y 1.522, Z 22.100}
   LaserEnd_Ext()
   LIN {X 7.993, Y 0.522, Z 22.100}
   LaserStart_Ext()
   LIN {X -2.781, Y 0.522, Z 22.100}
   LaserEnd_Ext()
   LIN {X -3.028, Y -0.478, Z 22.100}
   LaserStart_Ext()
   LIN {X 7.958, Y -0.478, Z 22.100}
   LaserEnd_Ext()
   LIN {X 7.924, Y -1.478, Z 22.100}
   LaserStart_Ext()
   LIN {X -3.340, Y -1.478, Z 22.100}
   LaserEnd_Ext()
   LIN {X -3.652, Y -2.478, Z 22.100}
   LaserStart_Ext()
   LIN {X 7.889, Y -2.478, Z 22.100}
   LaserEnd_Ext()
   LIN {X 7.845, Y -3.478, Z 22.100}
   LaserStart_Ext()
   LIN {X -3.963, Y -3.478, Z 22.100}
   LaserEnd_Ext()
   LIN {X -4.275, Y -4.478, Z 22.100}
   LaserStart_Ext()
   LIN {X 7.745, Y -4.478, Z 22.100}
   LaserEnd_Ext()
   LIN {X 7.635, Y -5.478, Z 22.100}
   LaserStart_Ext()
   LIN {X -4.587, Y -5.478, Z 22.100}
   LaserEnd_Ext()
   LIN {X -4.899, Y -6.478, Z 22.100}
   LaserStart_Ext()
   LIN {X 7.524, Y -6.478, Z 22.100}
   LaserEnd_Ext()
   LIN {X 7.413, Y -7.478, Z 22.100}
   LaserStart_Ext()
   LIN {X -5.297, Y -7.478, Z 22.100}
   LaserEnd_Ext()
   LIN {X -5.696, Y -8.478, Z 22.100}
   LaserStart_Ext()
   LIN {X 7.303, Y -8.478, Z 22.100}
   LaserEnd_Ext()
   LIN {X 7.192, Y -9.478, Z 22.100}
   LaserStart_Ext()
   LIN {X -6.095, Y -9.478, Z 22.100}
   LaserEnd_Ext()
   LIN {X -6.493, Y -10.478, Z 22.100}
   LaserStart_Ext()
   LIN {X 7.052, Y -10.478, Z 22.100}
   LaserEnd_Ext()
   LIN {X 6.894, Y -11.478, Z 22.100}
   LaserStart_Ext()
   LIN {X -6.925, Y -11.478, Z 22.100}
   LaserEnd_Ext()
   LIN {X -7.399, Y -12.478, Z 22.100}
   LaserStart_Ext()
   LIN {X 6.735, Y -12.478, Z 22.100}
   LaserEnd_Ext()
   LIN {X 6.568, Y -13.478, Z 22.100}
   LaserStart_Ext()
   LIN {X -7.876, Y -13.478, Z 22.100}
   LaserEnd_Ext()
   LIN {X -8.353, Y -14.478, Z 22.100}
   LaserStart_Ext()
   LIN {X 6.402, Y -14.478, Z 22.100}
   LaserEnd_Ext()
   LIN {X 6.216, Y -15.478, Z 22.100}
   LaserStart_Ext()
   LIN {X -8.845, Y -15.478, Z 22.100}
   LaserEnd_Ext()
   LIN {X -9.394, Y -16.478, Z 22.100}
   LaserStart_Ext()
   LIN {X 6.010, Y -16.478, Z 22.100}
   LaserEnd_Ext()
   LIN {X 5.804, Y -17.478, Z 22.100}
   LaserStart_Ext()
   LIN {X -0.891, Y -17.478, Z 22.100}
   LaserEnd_Ext()
   LIN {X -6.471, Y -17.478, Z 22.100}
   LaserStart_Ext()
   LIN {X -9.944, Y -17.478, Z 22.100}
   LaserEnd_Ext()
   LIN {X -10.493, Y -18.478, Z 22.100}
   LaserStart_Ext()
   LIN {X -7.875, Y -18.478, Z 22.100}
   LaserEnd_Ext()
   LIN {X 0.429, Y -18.478, Z 22.100}
   LaserStart_Ext()
   LIN {X 5.598, Y -18.478, Z 22.100}
   LaserEnd_Ext()
   LIN {X 5.370, Y -19.478, Z 22.100}
   LaserStart_Ext()
   LIN {X 1.201, Y -19.478, Z 22.100}
   LaserEnd_Ext()
   LIN {X -8.617, Y -19.478, Z 22.100}
   LaserStart_Ext()
   LIN {X -10.894, Y -19.478, Z 22.100}
   LaserEnd_Ext()
   LIN {X -11.263, Y -20.478, Z 22.100}
   LaserStart_Ext()
   LIN {X -9.130, Y -20.478, Z 22.100}
   LaserEnd_Ext()
   LIN {X 1.684, Y -20.478, Z 22.100}
   LaserStart_Ext()
   LIN {X 5.131, Y -20.478, Z 22.100}
   LaserEnd_Ext()
   LIN {X 4.893, Y -21.478, Z 22.100}
   LaserStart_Ext()
   LIN {X 2.152, Y -21.478, Z 22.100}
   LaserEnd_Ext()
   LIN {X -9.496, Y -21.478, Z 22.100}
   LaserStart_Ext()
   LIN {X -11.587, Y -21.478, Z 22.100}
   LaserEnd_Ext()
   LIN {X -11.555, Y -22.478, Z 22.100}
   LaserStart_Ext()
   LIN {X -9.712, Y -22.478, Z 22.100}
   LaserEnd_Ext()
   LIN {X 2.173, Y -22.478, Z 22.100}
   LaserStart_Ext()
   LIN {X 4.633, Y -22.478, Z 22.100}
   LaserEnd_Ext()
   LIN {X 4.366, Y -23.478, Z 22.100}
   LaserStart_Ext()
   LIN {X 2.144, Y -23.478, Z 22.100}
   LaserEnd_Ext()
   LIN {X -9.612, Y -23.478, Z 22.100}
   LaserStart_Ext()
   LIN {X -11.524, Y -23.478, Z 22.100}
   LaserEnd_Ext()
   LIN {X -11.498, Y -24.478, Z 22.100}
   LaserStart_Ext()
   LIN {X -9.477, Y -24.478, Z 22.100}
   LaserEnd_Ext()
   LIN {X 1.976, Y -24.478, Z 22.100}
   LaserStart_Ext()
   LIN {X 4.097, Y -24.478, Z 22.100}
   LaserEnd_Ext()
   LIN {X 3.688, Y -25.478, Z 22.100}
   LaserStart_Ext()
   LIN {X 1.475, Y -25.478, Z 22.100}
   LaserEnd_Ext()
   LIN {X -8.971, Y -25.478, Z 22.100}
   LaserStart_Ext()
   LIN {X -11.162, Y -25.478, Z 22.100}
   LaserEnd_Ext()
   LIN {X -10.735, Y -26.478, Z 22.100}
   LaserStart_Ext()
   LIN {X -8.403, Y -26.478, Z 22.100}
   LaserEnd_Ext()
   LIN {X 0.954, Y -26.478, Z 22.100}
   LaserStart_Ext()
   LIN {X 3.193, Y -26.478, Z 22.100}
   LaserEnd_Ext()
   LIN {X 2.651, Y -27.478, Z 22.100}
   LaserStart_Ext()
   LIN {X -0.287, Y -27.478, Z 22.100}
   LaserEnd_Ext()
   LIN {X -7.257, Y -27.478, Z 22.100}
   LaserStart_Ext()
   LIN {X -10.070, Y -27.478, Z 22.100}
   LaserEnd_Ext()
   LIN {X -9.092, Y -28.478, Z 22.100}
   LaserStart_Ext()
   LIN {X -5.119, Y -28.478, Z 22.100}
   LaserEnd_Ext()
   LIN {X -2.440, Y -28.478, Z 22.100}
   LaserStart_Ext()
   LIN {X 1.610, Y -28.478, Z 22.100}
   LaserEnd_Ext()
   LIN {X 0.349, Y -29.478, Z 22.100}
   LaserStart_Ext()
   LIN {X -8.016, Y -29.478, Z 22.100}
   LaserEnd_Ext()
   LIN {X -5.697, Y -30.478, Z 22.100}
   LaserStart_Ext()
   LIN {X -2.166, Y -30.478, Z 22.100}
   LaserEnd_Ext()
   LIN {X -0.410, Y -26.340, Z 22.950}
   LaserStart_Ext()
   LIN {X -1.625, Y -27.261, Z 22.950} C_DIS
   LIN {X -2.736, Y -27.489, Z 22.950} C_DIS
   LIN {X -3.747, Y -27.695, Z 22.950} C_DIS
   LIN {X -5.060, Y -27.402, Z 22.950} C_DIS
   LIN {X -5.759, Y -27.248, Z 22.950} C_DIS
   LIN {X -6.189, Y -26.929, Z 22.950} C_DIS
   LIN {X -7.413, Y -26.013, Z 22.950} C_DIS
   LIN {X -8.388, Y -24.299, Z 22.950} C_DIS
   LIN {X -8.429, Y -24.175, Z 22.950} C_DIS
   LIN {X -8.631, Y -22.337, Z 22.950} C_DIS
   LIN {X -8.466, Y -21.646, Z 22.950} C_DIS
   LIN {X -7.663, Y -20.079, Z 22.950} C_DIS
   LIN {X -7.312, Y -19.312, Z 22.950} C_DIS
   LIN {X -6.590, Y -18.800, Z 22.950} C_DIS
   LIN {X -5.609, Y -18.102, Z 22.950} C_DIS
   LIN {X -3.566, Y -17.694, Z 22.950} C_DIS
   LIN {X -2.039, Y -18.028, Z 22.950} C_DIS
   LIN {X -1.546, Y -18.137, Z 22.950} C_DIS
   LIN {X -1.206, Y -18.394, Z 22.950} C_DIS
   LIN {X 0.151, Y -19.415, Z 22.950} C_DIS
   LIN {X 1.106, Y -21.372, Z 22.950} C_DIS
   LIN {X 1.266, Y -21.701, Z 22.950} C_DIS
   LIN {X 1.255, Y -22.057, Z 22.950} C_DIS
   LIN {X 1.209, Y -23.876, Z 22.950} C_DIS
   LIN {X 0.468, Y -25.328, Z 22.950} C_DIS
   LIN {X 0.193, Y -25.876, Z 22.950} C_DIS
   LIN {X -0.410, Y -26.340, Z 22.950}
   LaserEnd_Ext()
   LIN {X 9.171, Y 4.544, Z 22.950}
   LaserStart_Ext()
   LIN {X 8.944, Y -1.979, Z 22.950} C_DIS
   LIN {X 8.861, Y -3.633, Z 22.950} C_DIS
   LIN {X 8.604, Y -6.163, Z 22.950} C_DIS
   LIN {X 8.199, Y -9.820, Z 22.950} C_DIS
   LIN {X 7.539, Y -14.003, Z 22.950} C_DIS
   LIN {X 7.350, Y -15.133, Z 22.950} C_DIS
   LIN {X 7.005, Y -16.810, Z 22.950} C_DIS
   LIN {X 6.571, Y -18.962, Z 22.950} C_DIS
   LIN {X 6.342, Y -19.949, Z 22.950} C_DIS
   LIN {X 5.866, Y -21.943, Z 22.950} C_DIS
   LIN {X 5.168, Y -24.551, Z 22.950} C_DIS
   LIN {X 5.025, Y -25.097, Z 22.950} C_DIS
   LIN {X 4.776, Y -25.565, Z 22.950} C_DIS
   LIN {X 3.503, Y -28.112, Z 22.950} C_DIS
   LIN {X 1.544, Y -29.994, Z 22.950} C_DIS
   LIN {X 1.368, Y -30.145, Z 22.950} C_DIS
   LIN {X 1.084, Y -30.247, Z 22.950} C_DIS
   LIN {X -2.379, Y -31.605, Z 22.950} C_DIS
   LIN {X -3.594, Y -31.572, Z 22.950} C_DIS
   LIN {X -5.348, Y -31.552, Z 22.950} C_DIS
   LIN {X -6.256, Y -31.300, Z 22.950} C_DIS
   LIN {X -8.338, Y -30.389, Z 22.950} C_DIS
   LIN {X -8.667, Y -30.209, Z 22.950} C_DIS
   LIN {X -8.912, Y -29.947, Z 22.950} C_DIS
   LIN {X -11.239, Y -27.607, Z 22.950} C_DIS
   LIN {X -12.224, Y -25.324, Z 22.950} C_DIS
   LIN {X -12.410, Y -24.886, Z 22.950} C_DIS
   LIN {X -12.421, Y -24.426, Z 22.950} C_DIS
   LIN {X -12.526, Y -21.177, Z 22.950} C_DIS
   LIN {X -11.755, Y -19.088, Z 22.950} C_DIS
   LIN {X -11.434, Y -18.201, Z 22.950} C_DIS
   LIN {X -10.651, Y -16.755, Z 22.950} C_DIS
   LIN {X -9.557, Y -14.764, Z 22.950} C_DIS
   LIN {X -8.642, Y -12.846, Z 22.950} C_DIS
   LIN {X -7.587, Y -10.601, Z 22.950} C_DIS
   LIN {X -6.681, Y -8.309, Z 22.950} C_DIS
   LIN {X -5.865, Y -6.265, Z 22.950} C_DIS
   LIN {X -4.746, Y -2.676, Z 22.950} C_DIS
   LIN {X -3.986, Y -0.251, Z 22.950} C_DIS
   LIN {X -3.255, Y 2.874, Z 22.950} C_DIS
   LIN {X -3.024, Y 3.856, Z 22.950} C_DIS
   LIN {X -2.945, Y 4.272, Z 22.950} C_DIS
   LIN {X -2.219, Y 8.576, Z 22.950} C_DIS
   LIN {X -2.103, Y 9.513, Z 22.950} C_DIS
   LIN {X -1.815, Y 12.246, Z 22.950} C_DIS
   LIN {X -1.697, Y 13.868, Z 22.950} C_DIS
   LIN {X -1.653, Y 16.637, Z 22.950} C_DIS
   LIN {X -1.620, Y 20.247, Z 22.950} C_DIS
   LIN {X -1.612, Y 21.320, Z 22.950} C_DIS
   LIN {X -2.011, Y 26.494, Z 22.950} C_DIS
   LIN {X -2.036, Y 26.792, Z 22.950} C_DIS
   LIN {X -2.274, Y 28.482, Z 22.950} C_DIS
   LIN {X -2.533, Y 30.331, Z 22.950} C_DIS
   LIN {X -2.611, Y 30.767, Z 22.950} C_DIS
   LIN {X -2.957, Y 32.664, Z 22.950} C_DIS
   LIN {X -3.444, Y 34.922, Z 22.950} C_DIS
   LIN {X -3.471, Y 35.037, Z 22.950} C_DIS
   LIN {X -3.838, Y 36.537, Z 22.950} C_DIS
   LIN {X -4.028, Y 37.276, Z 22.950} C_DIS
   LIN {X -4.151, Y 37.749, Z 22.950} C_DIS
   LIN {X -4.216, Y 38.368, Z 22.950} C_DIS
   LIN {X -4.288, Y 39.137, Z 22.950} C_DIS
   LIN {X -4.072, Y 39.913, Z 22.950} C_DIS
   LIN {X -3.877, Y 40.604, Z 22.950} C_DIS
   LIN {X -2.886, Y 41.735, Z 22.950} C_DIS
   LIN {X -2.596, Y 42.078, Z 22.950} C_DIS
   LIN {X -2.282, Y 42.181, Z 22.950} C_DIS
   LIN {X -0.319, Y 42.786, Z 22.950} C_DIS
   LIN {X 0.846, Y 42.521, Z 22.950} C_DIS
   LIN {X 1.384, Y 42.397, Z 22.950} C_DIS
   LIN {X 2.177, Y 41.778, Z 22.950} C_DIS
   LIN {X 2.757, Y 41.326, Z 22.950} C_DIS
   LIN {X 2.950, Y 40.981, Z 22.950} C_DIS
   LIN {X 3.472, Y 40.038, Z 22.950} C_DIS
   LIN {X 3.907, Y 38.706, Z 22.950} C_DIS
   LIN {X 3.960, Y 38.539, Z 22.950} C_DIS
   LIN {X 4.632, Y 36.355, Z 22.950} C_DIS
   LIN {X 5.025, Y 34.972, Z 22.950} C_DIS
   LIN {X 5.369, Y 33.750, Z 22.950} C_DIS
   LIN {X 5.579, Y 32.904, Z 22.950} C_DIS
   LIN {X 6.177, Y 30.555, Z 22.950} C_DIS
   LIN {X 6.727, Y 28.100, Z 22.950} C_DIS
   LIN {X 7.032, Y 26.665, Z 22.950} C_DIS
   LIN {X 7.570, Y 23.518, Z 22.950} C_DIS
   LIN {X 7.965, Y 21.287, Z 22.950} C_DIS
   LIN {X 8.289, Y 18.661, Z 22.950} C_DIS
   LIN {X 8.775, Y 14.489, Z 22.950} C_DIS
   LIN {X 8.928, Y 12.613, Z 22.950} C_DIS
   LIN {X 9.023, Y 10.264, Z 22.950} C_DIS
   LIN {X 9.171, Y 4.544, Z 22.950}
   LaserEnd_Ext()
   LIN {X -11.280, Y -24.989, Z 22.950}
   LaserStart_Ext()
   LIN {X -11.280, Y -20.688, Z 22.950}
   LaserEnd_Ext()
   LIN {X -10.280, Y -18.169, Z 22.950}
   LaserStart_Ext()
   LIN {X -10.280, Y -27.153, Z 22.950}
   LaserEnd_Ext()
   LIN {X -9.280, Y -28.159, Z 22.950}
   LaserStart_Ext()
   LIN {X -9.280, Y -24.754, Z 22.950}
   LaserEnd_Ext()
   LIN {X -9.280, Y -21.041, Z 22.950}
   LaserStart_Ext()
   LIN {X -9.280, Y -16.337, Z 22.950}
   LaserEnd_Ext()
   LIN {X -8.280, Y -14.410, Z 22.950}
   LaserStart_Ext()
   LIN {X -8.280, Y -19.024, Z 22.950}
   LaserEnd_Ext()
   LIN {X -8.280, Y -26.511, Z 22.950}
   LaserStart_Ext()
   LIN {X -8.280, Y -29.165, Z 22.950}
   LaserEnd_Ext()
   LIN {X -7.280, Y -29.760, Z 22.950}
   LaserStart_Ext()
   LIN {X -7.280, Y -27.362, Z 22.950}
   LaserEnd_Ext()
   LIN {X -7.280, Y -18.063, Z 22.950}
   LaserStart_Ext()
   LIN {X -7.280, Y -12.298, Z 22.950}
   LaserEnd_Ext()
   LIN {X -6.280, Y -10.014, Z 22.950}
   LaserStart_Ext()
   LIN {X -6.280, Y -17.352, Z 22.950}
   LaserEnd_Ext()
   LIN {X -6.280, Y -28.101, Z 22.950}
   LaserStart_Ext()
   LIN {X -6.280, Y -30.198, Z 22.950}
   LaserEnd_Ext()
   LIN {X -5.280, Y -30.533, Z 22.950}
   LaserStart_Ext()
   LIN {X -5.280, Y -28.378, Z 22.950}
   LaserEnd_Ext()
   LIN {X -5.280, Y -17.016, Z 22.950}
   LaserStart_Ext()
   LIN {X -5.280, Y -7.497, Z 22.950}
   LaserEnd_Ext()
   LIN {X -4.280, Y -4.541, Z 22.950}
   LaserStart_Ext()
   LIN {X -4.280, Y -16.817, Z 22.950}
   LaserEnd_Ext()
   LIN {X -4.280, Y -28.601, Z 22.950}
   LaserStart_Ext()
   LIN {X -4.280, Y -30.564, Z 22.950}
   LaserEnd_Ext()
   LIN {X -3.280, Y -30.580, Z 22.950}
   LaserStart_Ext()
   LIN {X -3.280, Y -28.621, Z 22.950}
   LaserEnd_Ext()
   LIN {X -3.280, Y -16.733, Z 22.950}
   LaserStart_Ext()
   LIN {X -3.280, Y -1.342, Z 22.950}
   LaserEnd_Ext()
   LIN {X -2.280, Y 40.910, Z 22.950}
   LaserStart_Ext()
   LIN {X -2.280, Y 34.266, Z 22.950}
   LaserEnd_Ext()
   LIN {X -2.280, Y 2.652, Z 22.950}
   LaserStart_Ext()
   LIN {X -2.280, Y -16.951, Z 22.950}
   LaserEnd_Ext()
   LIN {X -2.280, Y -28.416, Z 22.950}
   LaserStart_Ext()
   LIN {X -2.280, Y -30.492, Z 22.950}
   LaserEnd_Ext()
   LIN {X -1.280, Y -30.100, Z 22.950}
   LaserStart_Ext()
   LIN {X -1.280, Y -28.198, Z 22.950}
   LaserEnd_Ext()
   LIN {X -1.280, Y -17.175, Z 22.950}
   LaserStart_Ext()
   LIN {X -1.280, Y 8.129, Z 22.950}
   LaserEnd_Ext()
   LIN {X -1.280, Y 28.595, Z 22.950}
   LaserStart_Ext()
   LIN {X -1.280, Y 41.443, Z 22.950}
   LaserEnd_Ext()
   LIN {X -0.280, Y 41.752, Z 22.950}
   LaserStart_Ext()
   LIN {X -0.280, Y -17.840, Z 22.950}
   LaserEnd_Ext()
   LIN {X -0.280, Y -27.496, Z 22.950}
   LaserStart_Ext()
   LIN {X -0.280, Y -29.708, Z 22.950}
   LaserEnd_Ext()
   LIN {X 0.720, Y -29.316, Z 22.950}
   LaserStart_Ext()
   LIN {X 0.720, Y -26.732, Z 22.950}
   LaserEnd_Ext()
   LIN {X 0.720, Y -18.591, Z 22.950}
   LaserStart_Ext()
   LIN {X 0.720, Y 41.524, Z 22.950}
   LaserEnd_Ext()
   LIN {X 1.720, Y 40.866, Z 22.950}
   LaserStart_Ext()
   LIN {X 1.720, Y -20.350, Z 22.950}
   LaserEnd_Ext()
   LIN {X 1.720, Y -25.074, Z 22.950}
